// TIA Portal V19 export
// export: Created 2024-12-12T07:14:05.7970126Z, ExportSetting WithDefaults, DisplayName Totally Integrated Automation Portal, DisplayVersion V19 Update 1, DisplayName TIA Portal Openness, DisplayVersion V19 Update 1, DisplayName TIA Portal Version Control Interface, DisplayVersion V19, DisplayName SINAMICS Startdrive Advanced, DisplayVersion V19, DisplayName SINAMICS DCC, DisplayVersion V19, DisplayName SINAMICS Startdrive G130, G150, S120, S150, SINAMICS MV, G220, S200, S210, DisplayVersion V19, DisplayName SINAMICS Startdrive G110M, G120, G120C, G120D, G120P, G115D, DisplayVersion V19, DisplayName STEP 7 Professional, DisplayVersion V19 Update 1, DisplayName STEP 7 Safety, DisplayVersion V19 Update 1, DisplayName WinCC Advanced, DisplayVersion V19 Update 1, DisplayName WinCC Advanced / Unified PC, DisplayVersion V19 Update 1
DATA_BLOCK "AC1"   // DB1013
{ S7_Optimized_Access := 'TRUE' }
VERSION : 0.1
// stored: AutoNumber true, DBAccessibleFromOPCUA true, DBAccessibleFromWebserver true, InstanceOfName EM_AC120_1_2CG, InstanceOfType UDT, IsOnlyStoredInLoadMemory false, IsWriteProtectedInAS false
"EM_AC120_1_2CG"
   // VAR RETAIN
   //    Std : "EM_Std";
   //    Gen : "EM_AC120_1_2CG_Gen";
   //    Param : "EM_AC120_1_2CG_Param";
   //    LastHmiDataParam : "EM_AC120_1_2CG_Param";
   //    Alm : "EM_AC120_1_2CG_Alm";
   //    Sign : "EM_AC120_1_2CG_Sign";
   //    Input : "AC_Input";
   //    Output : "AC_Output";
   //    Ons : "AC_Ons";
   //    "Step" : "AC_Step";
   //    CamCalc : "EM_AC120_1_2CG_CamCalc";
   //    ExchangeFromChain : "EM_AC120_1_2CG_Exchange_FromChain";
   //    ExchangeToChain : "EM_AC120_1_2CG_Exchange_ToChain";
   //    Asc : "EM_AC120_1_2CG_Asc";
   //    Desc : "AC_AscDesc";
   //    Transfer : "EM_AC120_1_2CG_Transfer";
   //    VMaster : "EM_AC120_1_2CG_Virtual";
   //    ThermalReg1 : "AC_ThermalReg";
   //    ShiftUp : Array[0..127] of "TypeMouldData";
   //    ShiftTransfer : Array[0..127] of "TypeMouldData";
   //    ShiftDwn : Array[0..127] of "TypeMouldData";
   // END_VAR
BEGIN
   Std.Cfg_ModuleSync := TRUE;
   Std.Cfg_0_BelongShort_1_BelongLong := TRUE;
   Std.Cfg_ExternalCPU := FALSE;
   Std.Cfg_0_JogWord_1_JogBit := TRUE;
   Std._0_PriorityAlm_1_FirstAlm := FALSE;
   Std.AbortAlmOk := TRUE;
   Std.ServicesAbortAlmOk := TRUE;
   Std.SignOK := TRUE;
   Std.AlmReset := FALSE;
   Std.SignReset := FALSE;
   Std.NewAlm := FALSE;
   Std.NewSign := FALSE;
   Std.RstNewAlm := FALSE;
   Std.RstNewSign := FALSE;
   Std.AllowCopyByCategory := TRUE;
   Std.ForceCopyAll := FALSE;
   Std.InitCategories := FALSE;
   Std.InitCauses := FALSE;
   Std.Diag_AlmFound := FALSE;
   Std.Diag_SignFound := FALSE;
   Std.ScOk := FALSE;
   Std.OkToStop := TRUE;
   Std.PwrDrv := TRUE;
   Std.DriveRunCmd := FALSE;
   Std.ManAct := FALSE;
   Std.MachineSelected := TRUE;
   Std.MachineExtracted := FALSE;
   Std.LocalAbortReq := FALSE;
   Std.CondOkToEnaStaReq := FALSE;
   Std.EnaReq := FALSE;
   Std.EnaStaReq := FALSE;
   Std.StaReq := FALSE;
   Std.ReqStart := FALSE;
   Std.ReqStop := FALSE;
   Std.ReqAbort := TRUE;
   Std.ReqExecute := FALSE;
   Std.ReqReset := FALSE;
   Std.ReqSuspend := FALSE;
   Std.ReqUnSuspend := FALSE;
   Std.StrobeDeviceDiag := FALSE;
   Std.StrobeInverterDiag := FALSE;
   Std.DeviceDiagnosticDone := FALSE;
   Std.InverterDiagnosticDone := FALSE;
   Std.RecipeOnlineLoadDone := FALSE;
   Std.RecipeOnlineSaveDone := FALSE;
   Std.RecipeOfflineLoadDone := FALSE;
   Std.RecipeOfflineSaveDone := FALSE;
   Std.LastHmiDataLoadDone := FALSE;
   Std.LastHmiDataSaveDone := FALSE;
   Std.SummAlmTimeoutStart := FALSE;
   Std.SirenEna := FALSE;
   Std.VisEnButtons := TRUE;
   Std.VisManButtons := FALSE;
   Std.VisHomeButtons := FALSE;
   Std.VisEnButtonsRunning := TRUE;
   Std.Ena_Suspended := TRUE;
   Std.BluStkLgh_Steady_Cond := FALSE;
   Std.BluStkLgh_Frequency1_Cond := FALSE;
   Std.Siren_Frequency4_Cond := FALSE;
   Std.Cfg_ModuleNumber := 4;
   Std.Cfg_DeviceDiagCounter_Preset := 1;
   Std.Cfg_InverterDiagCounter_Preset := 1;
   Std.Cfg_Num_AlmDint := 11;
   Std.Cfg_Num_SignDint := 4;
   Std.Cfg_StaPbt := 65535;
   Std.Cfg_StoPbt := 65535;
   Std.Cfg_RstPbt := -1;
   Std.Cfg_EnaPbt := 65535;
   Std.Cfg_Siren := 1;
   Std.Cfg_Stack := 1;
   Std.Cfg_DisableStates[0..31] := 0;
   Std.Cfg_ModeTransitions[0..31] := 0;
   Std.Cfg_ModeNames[0..31] := '';
   Std.ModeCurrentName := 'Production';
   Std.StateCurrentName := 'Aborted';
   Std.DeviceDiagCounter := 0;
   Std.InverterDiagCounter := 0;
   Std.MaintenanceActivated."0" := FALSE;
   Std.MaintenanceActivated."1" := FALSE;
   Std.MaintenanceActivated."2" := FALSE;
   Std.MaintenanceActivated."3" := FALSE;
   Std.MaintenanceActivated."4" := FALSE;
   Std.MaintenanceActivated."5" := FALSE;
   Std.MaintenanceActivated."6" := FALSE;
   Std.MaintenanceActivated."7" := FALSE;
   Std.MaintenanceActivated."8" := FALSE;
   Std.MaintenanceActivated."9" := FALSE;
   Std.MaintenanceActivated."10" := FALSE;
   Std.MaintenanceActivated."11" := FALSE;
   Std.MaintenanceActivated."12" := FALSE;
   Std.MaintenanceActivated."13" := FALSE;
   Std.MaintenanceActivated."14" := FALSE;
   Std.MaintenanceActivated."15" := FALSE;
   Std.MaintenanceActivated."16" := FALSE;
   Std.MaintenanceActivated."17" := FALSE;
   Std.MaintenanceActivated."18" := FALSE;
   Std.MaintenanceActivated."19" := FALSE;
   Std.MaintenanceActivated."20" := FALSE;
   Std.MaintenanceActivated."21" := FALSE;
   Std.MaintenanceActivated."22" := FALSE;
   Std.MaintenanceActivated."23" := FALSE;
   Std.MaintenanceActivated."24" := FALSE;
   Std.MaintenanceActivated."25" := FALSE;
   Std.MaintenanceActivated."26" := FALSE;
   Std.MaintenanceActivated."27" := FALSE;
   Std.MaintenanceActivated."28" := FALSE;
   Std.MaintenanceActivated."29" := FALSE;
   Std.MaintenanceActivated."30" := FALSE;
   Std.MaintenanceActivated."31" := FALSE;
   Std.MaintenanceReq."0" := FALSE;
   Std.MaintenanceReq."1" := FALSE;
   Std.MaintenanceReq."2" := FALSE;
   Std.MaintenanceReq."3" := FALSE;
   Std.MaintenanceReq."4" := FALSE;
   Std.MaintenanceReq."5" := FALSE;
   Std.MaintenanceReq."6" := FALSE;
   Std.MaintenanceReq."7" := FALSE;
   Std.MaintenanceReq."8" := FALSE;
   Std.MaintenanceReq."9" := FALSE;
   Std.MaintenanceReq."10" := FALSE;
   Std.MaintenanceReq."11" := FALSE;
   Std.MaintenanceReq."12" := FALSE;
   Std.MaintenanceReq."13" := FALSE;
   Std.MaintenanceReq."14" := FALSE;
   Std.MaintenanceReq."15" := FALSE;
   Std.MaintenanceReq."16" := FALSE;
   Std.MaintenanceReq."17" := FALSE;
   Std.MaintenanceReq."18" := FALSE;
   Std.MaintenanceReq."19" := FALSE;
   Std.MaintenanceReq."20" := FALSE;
   Std.MaintenanceReq."21" := FALSE;
   Std.MaintenanceReq."22" := FALSE;
   Std.MaintenanceReq."23" := FALSE;
   Std.MaintenanceReq."24" := FALSE;
   Std.MaintenanceReq."25" := FALSE;
   Std.MaintenanceReq."26" := FALSE;
   Std.MaintenanceReq."27" := FALSE;
   Std.MaintenanceReq."28" := FALSE;
   Std.MaintenanceReq."29" := FALSE;
   Std.MaintenanceReq."30" := FALSE;
   Std.MaintenanceReq."31" := FALSE;
   Std.WithinScreenRange := 0;
   Std.ExchangeToGlobal.Communication.RunMode := FALSE;
   Std.ExchangeToGlobal.Communication.ConnectionFaulted := FALSE;
   Std.ExchangeToGlobal.Gen.Communication := FALSE;
   Std.ExchangeToGlobal.Gen.Selected := TRUE;
   Std.ExchangeToGlobal.Gen.Extracted := FALSE;
   Std.ExchangeToGlobal.Gen.EnaReq := FALSE;
   Std.ExchangeToGlobal.Gen.StaReq := FALSE;
   Std.ExchangeToGlobal.Gen.Started := FALSE;
   Std.ExchangeToGlobal.Gen.Unsuspended := FALSE;
   Std.ExchangeToGlobal.Gen.Ena_Suspended := TRUE;
   Std.ExchangeToGlobal.Gen.sts_Starting := FALSE;
   Std.ExchangeToGlobal.Gen.sts_Stopping := FALSE;
   Std.ExchangeToGlobal.Gen.sts_Aborting := FALSE;
   Std.ExchangeToGlobal.Gen.sts_Suspending := FALSE;
   Std.ExchangeToGlobal.Gen.sts_Unsuspending := FALSE;
   Std.ExchangeToGlobal.Gen.sts_Execute := FALSE;
   Std.ExchangeToGlobal.Gen.sts_Idle := FALSE;
   Std.ExchangeToGlobal.Gen.sts_Stopped := FALSE;
   Std.ExchangeToGlobal.Gen.sts_Aborted := TRUE;
   Std.ExchangeToGlobal.Gen.sts_Suspended := FALSE;
   Std.ExchangeToGlobal.Gen.sts_ModeManual := FALSE;
   Std.ExchangeToGlobal.Gen.sts_ModeAutomatic := TRUE;
   Std.ExchangeToGlobal.Gen.NewAlm := FALSE;
   Std.ExchangeToGlobal.Gen.NewSign := FALSE;
   Std.ExchangeToGlobal.Gen.RecipeOnlineLoadDone := FALSE;
   Std.ExchangeToGlobal.Gen.RecipeOnlineSaveDone := FALSE;
   Std.ExchangeToGlobal.Gen.RecipeOfflineLoadDone := FALSE;
   Std.ExchangeToGlobal.Gen.RecipeOfflineSaveDone := FALSE;
   Std.ExchangeToGlobal.Gen.LastHmiDataLoadDone := FALSE;
   Std.ExchangeToGlobal.Gen.LastHmiDataSaveDone := FALSE;
   Std.ExchangeToGlobal.Gen.InverterDiagnosticDone := FALSE;
   Std.ExchangeToGlobal.Gen.AxisGroupSync := TRUE;
   Std.ExchangeToGlobal.Gen.CmdMode := 1;
   Std.ExchangeToGlobal.Gen.Mode := 1;
   Std.ExchangeToGlobal.Gen.DisableEnaPbt := 0;
   Std.ExchangeToGlobal.Input.StaPbt := FALSE;
   Std.ExchangeToGlobal.Input.StoPbt := FALSE;
   Std.ExchangeToGlobal.Input.RstPbt := FALSE;
   Std.ExchangeToGlobal.Input.EnaPbt := FALSE;
   Std.ExchangeToGlobal.Input._4 := FALSE;
   Std.ExchangeToGlobal.Input._5 := FALSE;
   Std.ExchangeToGlobal.Input._6 := FALSE;
   Std.ExchangeToGlobal.Input._7 := FALSE;
   Std.ExchangeToGlobal.Input._8 := FALSE;
   Std.ExchangeToGlobal.Input._9 := FALSE;
   Std.ExchangeToGlobal.Input._10 := FALSE;
   Std.ExchangeToGlobal.Input._11 := FALSE;
   Std.ExchangeToGlobal.Input._12 := FALSE;
   Std.ExchangeToGlobal.Input._13 := FALSE;
   Std.ExchangeToGlobal.Input._14 := FALSE;
   Std.ExchangeToGlobal.Input._15 := FALSE;
   Std.ExchangeToGlobal.AlmOk.ThSwitch := TRUE;
   Std.ExchangeToGlobal.AlmOk.SafeComm := TRUE;
   Std.ExchangeToGlobal.AlmOk.SafeEmg := TRUE;
   Std.ExchangeToGlobal.AlmOk.SafeGuards := TRUE;
   Std.ExchangeToGlobal.AlmOk.GtaAirGroup := TRUE;
   Std.ExchangeToGlobal.AlmOk.Major := TRUE;
   Std.ExchangeToGlobal.AlmOk.Minor := TRUE;
   Std.ExchangeToGlobal.AlmOk.Spare07 := TRUE;
   Std.ExchangeToGlobal.AlmOk.Spare08 := TRUE;
   Std.ExchangeToGlobal.AlmOk.Spare09 := TRUE;
   Std.ExchangeToGlobal.AlmOk.Spare10 := TRUE;
   Std.ExchangeToGlobal.AlmOk.Spare11 := TRUE;
   Std.ExchangeToGlobal.AlmOk.Spare12 := TRUE;
   Std.ExchangeToGlobal.AlmOk.Spare13 := TRUE;
   Std.ExchangeToGlobal.AlmOk.Spare14 := TRUE;
   Std.ExchangeToGlobal.AlmOk.Spare15 := TRUE;
   Std.ExchangeToGlobal.AlmOk.Spare16 := TRUE;
   Std.ExchangeToGlobal.AlmOk.Spare17 := TRUE;
   Std.ExchangeToGlobal.AlmOk.Spare18 := TRUE;
   Std.ExchangeToGlobal.AlmOk.Spare19 := TRUE;
   Std.ExchangeToGlobal.AlmOk.Spare20 := TRUE;
   Std.ExchangeToGlobal.AlmOk.Spare21 := TRUE;
   Std.ExchangeToGlobal.AlmOk.Spare22 := TRUE;
   Std.ExchangeToGlobal.AlmOk.Spare23 := TRUE;
   Std.ExchangeToGlobal.AlmOk.Spare24 := TRUE;
   Std.ExchangeToGlobal.AlmOk.Spare25 := TRUE;
   Std.ExchangeToGlobal.AlmOk.Spare26 := TRUE;
   Std.ExchangeToGlobal.AlmOk.Spare27 := TRUE;
   Std.ExchangeToGlobal.AlmOk.Spare28 := TRUE;
   Std.ExchangeToGlobal.AlmOk.Spare29 := TRUE;
   Std.ExchangeToGlobal.AlmOk.Spare30 := TRUE;
   Std.ExchangeToGlobal.AlmOk.Spare31 := TRUE;
   Std.ExchangeToGlobal.AlmCauseOk.Ope := TRUE;
   Std.ExchangeToGlobal.AlmCauseOk.Ust := TRUE;
   Std.ExchangeToGlobal.AlmCauseOk.Dst := TRUE;
   Std.ExchangeToGlobal.AlmCauseOk.Ext := TRUE;
   Std.ExchangeToGlobal.AlmCauseOk.Mac := TRUE;
   Std.ExchangeToGlobal.AlmCauseOk.Spare05 := TRUE;
   Std.ExchangeToGlobal.AlmCauseOk.Spare06 := TRUE;
   Std.ExchangeToGlobal.AlmCauseOk.Spare07 := TRUE;
   Std.ExchangeToGlobal.AlmCauseOk.Spare08 := TRUE;
   Std.ExchangeToGlobal.AlmCauseOk.Spare09 := TRUE;
   Std.ExchangeToGlobal.AlmCauseOk.Spare10 := TRUE;
   Std.ExchangeToGlobal.AlmCauseOk.Spare11 := TRUE;
   Std.ExchangeToGlobal.AlmCauseOk.Spare12 := TRUE;
   Std.ExchangeToGlobal.AlmCauseOk.Spare13 := TRUE;
   Std.ExchangeToGlobal.AlmCauseOk.Spare14 := TRUE;
   Std.ExchangeToGlobal.AlmCauseOk.Spare15 := TRUE;
   Std.ExchangeToGlobal.AlmCauseOk.Spare16 := TRUE;
   Std.ExchangeToGlobal.AlmCauseOk.Spare17 := TRUE;
   Std.ExchangeToGlobal.AlmCauseOk.Spare18 := TRUE;
   Std.ExchangeToGlobal.AlmCauseOk.Spare19 := TRUE;
   Std.ExchangeToGlobal.AlmCauseOk.Spare20 := TRUE;
   Std.ExchangeToGlobal.AlmCauseOk.Spare21 := TRUE;
   Std.ExchangeToGlobal.AlmCauseOk.Spare22 := TRUE;
   Std.ExchangeToGlobal.AlmCauseOk.Spare23 := TRUE;
   Std.ExchangeToGlobal.AlmCauseOk.Spare24 := TRUE;
   Std.ExchangeToGlobal.AlmCauseOk.Spare25 := TRUE;
   Std.ExchangeToGlobal.AlmCauseOk.Spare26 := TRUE;
   Std.ExchangeToGlobal.AlmCauseOk.Spare27 := TRUE;
   Std.ExchangeToGlobal.AlmCauseOk.Spare28 := TRUE;
   Std.ExchangeToGlobal.AlmCauseOk.Spare29 := TRUE;
   Std.ExchangeToGlobal.AlmCauseOk.Spare30 := TRUE;
   Std.ExchangeToGlobal.AlmCauseOk.Spare31 := TRUE;
   Std.ExchangeToGlobal.AlmBannerFbk.FirstAlmDetection := FALSE;
   Std.ExchangeToGlobal.AlmBannerFbk.AlmPriority := 100;
   Std.ExchangeToGlobal.AlmBannerFbk.AlmCategory := -1;
   Std.ExchangeToGlobal.AlmBannerFbk.AlmCause := -1;
   Std.ExchangeToGlobal.AlmBannerFbk.AlmID := -1;
   Std.ExchangeToGlobal.AlmBannerFbk.GlobalAbsTime := 0;
   Std.ExchangeToGlobal.SignBannerFbk.SignPriority := 100;
   Std.ExchangeToGlobal.SignBannerFbk.SignCategory := -1;
   Std.ExchangeToGlobal.SignBannerFbk.SignID := -1;
   Std.ExchangeToGlobal.ExtCPU.PushButton.StaPbt := FALSE;
   Std.ExchangeToGlobal.ExtCPU.PushButton.StoPbt := FALSE;
   Std.ExchangeToGlobal.ExtCPU.PushButton.RstPbt := FALSE;
   Std.ExchangeToGlobal.ExtCPU.PushButton.EnaPbt := FALSE;
   Std.ExchangeToGlobal.ExtCPU.PushButton.EnaReq := FALSE;
   Std.ExchangeToGlobal.ExtCPU.PushButton.EnaStaReq := FALSE;
   Std.ExchangeToGlobal.ExtCPU.DeviceDiagDone := FALSE;
   Std.ExchangeToGlobal.ExtCPU.InverterDiagDone := FALSE;
   Std.ExchangeToGlobal.LightSiren.Cfg_StaPbt := 65535;
   Std.ExchangeToGlobal.LightSiren.Cfg_RstPbt := -1;
   Std.ExchangeToGlobal.LightSiren.Cfg_EnaPbt := 65535;
   Std.ExchangeToGlobal.LightSiren.Cfg_Siren := 1;
   Std.ExchangeToGlobal.LightSiren.Cfg_Stack := 1;
   Std.ExchangeToGlobal.LightSiren.Steady.StaPbtLgh := FALSE;
   Std.ExchangeToGlobal.LightSiren.Steady.RstPbtLgh := FALSE;
   Std.ExchangeToGlobal.LightSiren.Steady.EnaPbtLgh := FALSE;
   Std.ExchangeToGlobal.LightSiren.Steady.Siren := FALSE;
   Std.ExchangeToGlobal.LightSiren.Steady.YelStkLgh := FALSE;
   Std.ExchangeToGlobal.LightSiren.Steady.BluStkLgh := FALSE;
   Std.ExchangeToGlobal.LightSiren.Steady.GrnStkLgh := FALSE;
   Std.ExchangeToGlobal.LightSiren.Steady.WhtStkLgh := FALSE;
   Std.ExchangeToGlobal.LightSiren.Steady.Cust1_StaPbtLgh := FALSE;
   Std.ExchangeToGlobal.LightSiren.Steady.Cust1_RstPbtLgh := FALSE;
   Std.ExchangeToGlobal.LightSiren.Steady.Cust1_Siren := FALSE;
   Std.ExchangeToGlobal.LightSiren.Steady.Cust1_RedStkLgh := FALSE;
   Std.ExchangeToGlobal.LightSiren.Steady.Cust1_OngStkLgh := FALSE;
   Std.ExchangeToGlobal.LightSiren.Steady.Cust1_GrnStkLgh := FALSE;
   Std.ExchangeToGlobal.LightSiren.Steady.Cust1_BluStkLgh := FALSE;
   Std.ExchangeToGlobal.LightSiren.Steady.Cust1_WhtStkLgh := FALSE;
   Std.ExchangeToGlobal.LightSiren.Frequency1.StaPbtLgh := FALSE;
   Std.ExchangeToGlobal.LightSiren.Frequency1.RstPbtLgh := FALSE;
   Std.ExchangeToGlobal.LightSiren.Frequency1.EnaPbtLgh := FALSE;
   Std.ExchangeToGlobal.LightSiren.Frequency1.Siren := FALSE;
   Std.ExchangeToGlobal.LightSiren.Frequency1.YelStkLgh := FALSE;
   Std.ExchangeToGlobal.LightSiren.Frequency1.BluStkLgh := FALSE;
   Std.ExchangeToGlobal.LightSiren.Frequency1.GrnStkLgh := FALSE;
   Std.ExchangeToGlobal.LightSiren.Frequency1.WhtStkLgh := FALSE;
   Std.ExchangeToGlobal.LightSiren.Frequency1.Cust1_StaPbtLgh := FALSE;
   Std.ExchangeToGlobal.LightSiren.Frequency1.Cust1_RstPbtLgh := FALSE;
   Std.ExchangeToGlobal.LightSiren.Frequency1.Cust1_Siren := FALSE;
   Std.ExchangeToGlobal.LightSiren.Frequency1.Cust1_RedStkLgh := FALSE;
   Std.ExchangeToGlobal.LightSiren.Frequency1.Cust1_OngStkLgh := FALSE;
   Std.ExchangeToGlobal.LightSiren.Frequency1.Cust1_GrnStkLgh := FALSE;
   Std.ExchangeToGlobal.LightSiren.Frequency1.Cust1_BluStkLgh := FALSE;
   Std.ExchangeToGlobal.LightSiren.Frequency1.Cust1_WhtStkLgh := FALSE;
   Std.ExchangeToGlobal.LightSiren.Frequency2.StaPbtLgh := FALSE;
   Std.ExchangeToGlobal.LightSiren.Frequency2.RstPbtLgh := FALSE;
   Std.ExchangeToGlobal.LightSiren.Frequency2.EnaPbtLgh := FALSE;
   Std.ExchangeToGlobal.LightSiren.Frequency2.Siren := FALSE;
   Std.ExchangeToGlobal.LightSiren.Frequency2.YelStkLgh := FALSE;
   Std.ExchangeToGlobal.LightSiren.Frequency2.BluStkLgh := FALSE;
   Std.ExchangeToGlobal.LightSiren.Frequency2.GrnStkLgh := FALSE;
   Std.ExchangeToGlobal.LightSiren.Frequency2.WhtStkLgh := FALSE;
   Std.ExchangeToGlobal.LightSiren.Frequency2.Cust1_StaPbtLgh := FALSE;
   Std.ExchangeToGlobal.LightSiren.Frequency2.Cust1_RstPbtLgh := FALSE;
   Std.ExchangeToGlobal.LightSiren.Frequency2.Cust1_Siren := FALSE;
   Std.ExchangeToGlobal.LightSiren.Frequency2.Cust1_RedStkLgh := FALSE;
   Std.ExchangeToGlobal.LightSiren.Frequency2.Cust1_OngStkLgh := FALSE;
   Std.ExchangeToGlobal.LightSiren.Frequency2.Cust1_GrnStkLgh := FALSE;
   Std.ExchangeToGlobal.LightSiren.Frequency2.Cust1_BluStkLgh := FALSE;
   Std.ExchangeToGlobal.LightSiren.Frequency2.Cust1_WhtStkLgh := FALSE;
   Std.ExchangeToGlobal.LightSiren.Frequency3.StaPbtLgh := FALSE;
   Std.ExchangeToGlobal.LightSiren.Frequency3.RstPbtLgh := FALSE;
   Std.ExchangeToGlobal.LightSiren.Frequency3.EnaPbtLgh := FALSE;
   Std.ExchangeToGlobal.LightSiren.Frequency3.Siren := FALSE;
   Std.ExchangeToGlobal.LightSiren.Frequency3.YelStkLgh := FALSE;
   Std.ExchangeToGlobal.LightSiren.Frequency3.BluStkLgh := FALSE;
   Std.ExchangeToGlobal.LightSiren.Frequency3.GrnStkLgh := FALSE;
   Std.ExchangeToGlobal.LightSiren.Frequency3.WhtStkLgh := FALSE;
   Std.ExchangeToGlobal.LightSiren.Frequency3.Cust1_StaPbtLgh := FALSE;
   Std.ExchangeToGlobal.LightSiren.Frequency3.Cust1_RstPbtLgh := FALSE;
   Std.ExchangeToGlobal.LightSiren.Frequency3.Cust1_Siren := FALSE;
   Std.ExchangeToGlobal.LightSiren.Frequency3.Cust1_RedStkLgh := FALSE;
   Std.ExchangeToGlobal.LightSiren.Frequency3.Cust1_OngStkLgh := FALSE;
   Std.ExchangeToGlobal.LightSiren.Frequency3.Cust1_GrnStkLgh := FALSE;
   Std.ExchangeToGlobal.LightSiren.Frequency3.Cust1_BluStkLgh := FALSE;
   Std.ExchangeToGlobal.LightSiren.Frequency3.Cust1_WhtStkLgh := FALSE;
   Std.ExchangeToGlobal.LightSiren.Frequency4.StaPbtLgh := FALSE;
   Std.ExchangeToGlobal.LightSiren.Frequency4.RstPbtLgh := FALSE;
   Std.ExchangeToGlobal.LightSiren.Frequency4.EnaPbtLgh := FALSE;
   Std.ExchangeToGlobal.LightSiren.Frequency4.Siren := FALSE;
   Std.ExchangeToGlobal.LightSiren.Frequency4.YelStkLgh := FALSE;
   Std.ExchangeToGlobal.LightSiren.Frequency4.BluStkLgh := FALSE;
   Std.ExchangeToGlobal.LightSiren.Frequency4.GrnStkLgh := FALSE;
   Std.ExchangeToGlobal.LightSiren.Frequency4.WhtStkLgh := FALSE;
   Std.ExchangeToGlobal.LightSiren.Frequency4.Cust1_StaPbtLgh := FALSE;
   Std.ExchangeToGlobal.LightSiren.Frequency4.Cust1_RstPbtLgh := FALSE;
   Std.ExchangeToGlobal.LightSiren.Frequency4.Cust1_Siren := FALSE;
   Std.ExchangeToGlobal.LightSiren.Frequency4.Cust1_RedStkLgh := FALSE;
   Std.ExchangeToGlobal.LightSiren.Frequency4.Cust1_OngStkLgh := FALSE;
   Std.ExchangeToGlobal.LightSiren.Frequency4.Cust1_GrnStkLgh := FALSE;
   Std.ExchangeToGlobal.LightSiren.Frequency4.Cust1_BluStkLgh := FALSE;
   Std.ExchangeToGlobal.LightSiren.Frequency4.Cust1_WhtStkLgh := FALSE;
   Std.ExchangeToGlobal.PackML.Sts_Aborted := TRUE;
   Std.ExchangeToGlobal.PackML.Sts_Aborting := FALSE;
   Std.ExchangeToGlobal.PackML.Sts_Clearing := FALSE;
   Std.ExchangeToGlobal.PackML.Sts_Complete := FALSE;
   Std.ExchangeToGlobal.PackML.Sts_Completing := FALSE;
   Std.ExchangeToGlobal.PackML.Sts_Execute := FALSE;
   Std.ExchangeToGlobal.PackML.Sts_Held := FALSE;
   Std.ExchangeToGlobal.PackML.Sts_Holding := FALSE;
   Std.ExchangeToGlobal.PackML.Sts_Idle := FALSE;
   Std.ExchangeToGlobal.PackML.Sts_Resetting := FALSE;
   Std.ExchangeToGlobal.PackML.Sts_Starting := FALSE;
   Std.ExchangeToGlobal.PackML.Sts_Stopped := FALSE;
   Std.ExchangeToGlobal.PackML.Sts_Stopping := FALSE;
   Std.ExchangeToGlobal.PackML.Sts_Suspended := FALSE;
   Std.ExchangeToGlobal.PackML.Sts_Suspending := FALSE;
   Std.ExchangeToGlobal.PackML.Sts_UnHolding := FALSE;
   Std.ExchangeToGlobal.PackML.Sts_UnSuspending := FALSE;
   Std.ExchangeToGlobal.PackML.Sts_AbortedEnabled := TRUE;
   Std.ExchangeToGlobal.PackML.Sts_AbortingEnabled := TRUE;
   Std.ExchangeToGlobal.PackML.Sts_ClearingEnabled := TRUE;
   Std.ExchangeToGlobal.PackML.Sts_CompleteEnabled := FALSE;
   Std.ExchangeToGlobal.PackML.Sts_CompletingEnabled := FALSE;
   Std.ExchangeToGlobal.PackML.Sts_ExecuteEnabled := TRUE;
   Std.ExchangeToGlobal.PackML.Sts_HeldEnabled := FALSE;
   Std.ExchangeToGlobal.PackML.Sts_HoldingEnabled := FALSE;
   Std.ExchangeToGlobal.PackML.Sts_IdleEnabled := TRUE;
   Std.ExchangeToGlobal.PackML.Sts_ResettingEnabled := TRUE;
   Std.ExchangeToGlobal.PackML.Sts_StartingEnabled := TRUE;
   Std.ExchangeToGlobal.PackML.Sts_StoppedEnabled := TRUE;
   Std.ExchangeToGlobal.PackML.Sts_StoppingEnabled := TRUE;
   Std.ExchangeToGlobal.PackML.Sts_SuspendedEnabled := TRUE;
   Std.ExchangeToGlobal.PackML.Sts_SuspendingEnabled := TRUE;
   Std.ExchangeToGlobal.PackML.Sts_UnHoldingEnabled := FALSE;
   Std.ExchangeToGlobal.PackML.Sts_UnSuspendingEnabled := TRUE;
   Std.ExchangeToGlobal.SignOk := TRUE;
   Std.ExchangeToGlobal."Dint"[0..4] := 0;
   Std.VisAlmTypeBool.ThSwitch := FALSE;
   Std.VisAlmTypeBool.SafeComm := FALSE;
   Std.VisAlmTypeBool.SafeEmg := FALSE;
   Std.VisAlmTypeBool.SafeGuards := TRUE;
   Std.VisAlmTypeBool.GtaAirGroup := FALSE;
   Std.VisAlmTypeBool.Major := FALSE;
   Std.VisAlmTypeBool.Minor := FALSE;
   Std.VisAlmTypeBool.Spare07 := FALSE;
   Std.VisAlmTypeBool.Spare08 := FALSE;
   Std.VisAlmTypeBool.Spare09 := FALSE;
   Std.VisAlmTypeBool.Spare10 := FALSE;
   Std.VisAlmTypeBool.Spare11 := FALSE;
   Std.VisAlmTypeBool.Spare12 := FALSE;
   Std.VisAlmTypeBool.Spare13 := FALSE;
   Std.VisAlmTypeBool.Spare14 := FALSE;
   Std.VisAlmTypeBool.Spare15 := FALSE;
   Std.VisAlmTypeBool.Spare16 := FALSE;
   Std.VisAlmTypeBool.Spare17 := FALSE;
   Std.VisAlmTypeBool.Spare18 := FALSE;
   Std.VisAlmTypeBool.Spare19 := FALSE;
   Std.VisAlmTypeBool.Spare20 := FALSE;
   Std.VisAlmTypeBool.Spare21 := FALSE;
   Std.VisAlmTypeBool.Spare22 := FALSE;
   Std.VisAlmTypeBool.Spare23 := FALSE;
   Std.VisAlmTypeBool.Spare24 := FALSE;
   Std.VisAlmTypeBool.Spare25 := FALSE;
   Std.VisAlmTypeBool.Spare26 := FALSE;
   Std.VisAlmTypeBool.Spare27 := FALSE;
   Std.VisAlmTypeBool.Spare28 := FALSE;
   Std.VisAlmTypeBool.Spare29 := FALSE;
   Std.VisAlmTypeBool.Spare30 := FALSE;
   Std.VisAlmTypeBool.Spare31 := FALSE;
   Std.AlmTypeFbk.ThSwitch := FALSE;
   Std.AlmTypeFbk.SafeComm := FALSE;
   Std.AlmTypeFbk.SafeEmg := FALSE;
   Std.AlmTypeFbk.SafeGuards := FALSE;
   Std.AlmTypeFbk.GtaAirGroup := FALSE;
   Std.AlmTypeFbk.Major := FALSE;
   Std.AlmTypeFbk.Minor := FALSE;
   Std.AlmTypeFbk.Spare07 := FALSE;
   Std.AlmTypeFbk.Spare08 := FALSE;
   Std.AlmTypeFbk.Spare09 := FALSE;
   Std.AlmTypeFbk.Spare10 := FALSE;
   Std.AlmTypeFbk.Spare11 := FALSE;
   Std.AlmTypeFbk.Spare12 := FALSE;
   Std.AlmTypeFbk.Spare13 := FALSE;
   Std.AlmTypeFbk.Spare14 := FALSE;
   Std.AlmTypeFbk.Spare15 := FALSE;
   Std.AlmTypeFbk.Spare16 := FALSE;
   Std.AlmTypeFbk.Spare17 := FALSE;
   Std.AlmTypeFbk.Spare18 := FALSE;
   Std.AlmTypeFbk.Spare19 := FALSE;
   Std.AlmTypeFbk.Spare20 := FALSE;
   Std.AlmTypeFbk.Spare21 := FALSE;
   Std.AlmTypeFbk.Spare22 := FALSE;
   Std.AlmTypeFbk.Spare23 := FALSE;
   Std.AlmTypeFbk.Spare24 := FALSE;
   Std.AlmTypeFbk.Spare25 := FALSE;
   Std.AlmTypeFbk.Spare26 := FALSE;
   Std.AlmTypeFbk.Spare27 := FALSE;
   Std.AlmTypeFbk.Spare28 := FALSE;
   Std.AlmTypeFbk.Spare29 := FALSE;
   Std.AlmTypeFbk.Spare30 := FALSE;
   Std.AlmTypeFbk.Spare31 := FALSE;
   Std.AlmTypeOk.ThSwitch := TRUE;
   Std.AlmTypeOk.SafeComm := TRUE;
   Std.AlmTypeOk.SafeEmg := TRUE;
   Std.AlmTypeOk.SafeGuards := TRUE;
   Std.AlmTypeOk.GtaAirGroup := TRUE;
   Std.AlmTypeOk.Major := TRUE;
   Std.AlmTypeOk.Minor := TRUE;
   Std.AlmTypeOk.Spare07 := TRUE;
   Std.AlmTypeOk.Spare08 := TRUE;
   Std.AlmTypeOk.Spare09 := TRUE;
   Std.AlmTypeOk.Spare10 := TRUE;
   Std.AlmTypeOk.Spare11 := TRUE;
   Std.AlmTypeOk.Spare12 := TRUE;
   Std.AlmTypeOk.Spare13 := TRUE;
   Std.AlmTypeOk.Spare14 := TRUE;
   Std.AlmTypeOk.Spare15 := TRUE;
   Std.AlmTypeOk.Spare16 := TRUE;
   Std.AlmTypeOk.Spare17 := TRUE;
   Std.AlmTypeOk.Spare18 := TRUE;
   Std.AlmTypeOk.Spare19 := TRUE;
   Std.AlmTypeOk.Spare20 := TRUE;
   Std.AlmTypeOk.Spare21 := TRUE;
   Std.AlmTypeOk.Spare22 := TRUE;
   Std.AlmTypeOk.Spare23 := TRUE;
   Std.AlmTypeOk.Spare24 := TRUE;
   Std.AlmTypeOk.Spare25 := TRUE;
   Std.AlmTypeOk.Spare26 := TRUE;
   Std.AlmTypeOk.Spare27 := TRUE;
   Std.AlmTypeOk.Spare28 := TRUE;
   Std.AlmTypeOk.Spare29 := TRUE;
   Std.AlmTypeOk.Spare30 := TRUE;
   Std.AlmTypeOk.Spare31 := TRUE;
   Std.AlmCauseFbk.Ope := FALSE;
   Std.AlmCauseFbk.Ust := FALSE;
   Std.AlmCauseFbk.Dst := FALSE;
   Std.AlmCauseFbk.Ext := FALSE;
   Std.AlmCauseFbk.Mac := FALSE;
   Std.AlmCauseFbk.Spare05 := FALSE;
   Std.AlmCauseFbk.Spare06 := FALSE;
   Std.AlmCauseFbk.Spare07 := FALSE;
   Std.AlmCauseFbk.Spare08 := FALSE;
   Std.AlmCauseFbk.Spare09 := FALSE;
   Std.AlmCauseFbk.Spare10 := FALSE;
   Std.AlmCauseFbk.Spare11 := FALSE;
   Std.AlmCauseFbk.Spare12 := FALSE;
   Std.AlmCauseFbk.Spare13 := FALSE;
   Std.AlmCauseFbk.Spare14 := FALSE;
   Std.AlmCauseFbk.Spare15 := FALSE;
   Std.AlmCauseFbk.Spare16 := FALSE;
   Std.AlmCauseFbk.Spare17 := FALSE;
   Std.AlmCauseFbk.Spare18 := FALSE;
   Std.AlmCauseFbk.Spare19 := FALSE;
   Std.AlmCauseFbk.Spare20 := FALSE;
   Std.AlmCauseFbk.Spare21 := FALSE;
   Std.AlmCauseFbk.Spare22 := FALSE;
   Std.AlmCauseFbk.Spare23 := FALSE;
   Std.AlmCauseFbk.Spare24 := FALSE;
   Std.AlmCauseFbk.Spare25 := FALSE;
   Std.AlmCauseFbk.Spare26 := FALSE;
   Std.AlmCauseFbk.Spare27 := FALSE;
   Std.AlmCauseFbk.Spare28 := FALSE;
   Std.AlmCauseFbk.Spare29 := FALSE;
   Std.AlmCauseFbk.Spare30 := FALSE;
   Std.AlmCauseFbk.Spare31 := FALSE;
   Std.AlmCauseOk.Ope := TRUE;
   Std.AlmCauseOk.Ust := TRUE;
   Std.AlmCauseOk.Dst := TRUE;
   Std.AlmCauseOk.Ext := TRUE;
   Std.AlmCauseOk.Mac := TRUE;
   Std.AlmCauseOk.Spare05 := TRUE;
   Std.AlmCauseOk.Spare06 := TRUE;
   Std.AlmCauseOk.Spare07 := TRUE;
   Std.AlmCauseOk.Spare08 := TRUE;
   Std.AlmCauseOk.Spare09 := TRUE;
   Std.AlmCauseOk.Spare10 := TRUE;
   Std.AlmCauseOk.Spare11 := TRUE;
   Std.AlmCauseOk.Spare12 := TRUE;
   Std.AlmCauseOk.Spare13 := TRUE;
   Std.AlmCauseOk.Spare14 := TRUE;
   Std.AlmCauseOk.Spare15 := TRUE;
   Std.AlmCauseOk.Spare16 := TRUE;
   Std.AlmCauseOk.Spare17 := TRUE;
   Std.AlmCauseOk.Spare18 := TRUE;
   Std.AlmCauseOk.Spare19 := TRUE;
   Std.AlmCauseOk.Spare20 := TRUE;
   Std.AlmCauseOk.Spare21 := TRUE;
   Std.AlmCauseOk.Spare22 := TRUE;
   Std.AlmCauseOk.Spare23 := TRUE;
   Std.AlmCauseOk.Spare24 := TRUE;
   Std.AlmCauseOk.Spare25 := TRUE;
   Std.AlmCauseOk.Spare26 := TRUE;
   Std.AlmCauseOk.Spare27 := TRUE;
   Std.AlmCauseOk.Spare28 := TRUE;
   Std.AlmCauseOk.Spare29 := TRUE;
   Std.AlmCauseOk.Spare30 := TRUE;
   Std.AlmCauseOk.Spare31 := TRUE;
   Std.ForceCategory.ThSwitch := FALSE;
   Std.ForceCategory.SafeComm := TRUE;
   Std.ForceCategory.SafeEmg := TRUE;
   Std.ForceCategory.SafeGuards := FALSE;
   Std.ForceCategory.GtaAirGroup := FALSE;
   Std.ForceCategory.Major := FALSE;
   Std.ForceCategory.Minor := FALSE;
   Std.ForceCategory.Spare07 := FALSE;
   Std.ForceCategory.Spare08 := FALSE;
   Std.ForceCategory.Spare09 := FALSE;
   Std.ForceCategory.Spare10 := FALSE;
   Std.ForceCategory.Spare11 := FALSE;
   Std.ForceCategory.Spare12 := FALSE;
   Std.ForceCategory.Spare13 := FALSE;
   Std.ForceCategory.Spare14 := FALSE;
   Std.ForceCategory.Spare15 := FALSE;
   Std.ForceCategory.Spare16 := FALSE;
   Std.ForceCategory.Spare17 := FALSE;
   Std.ForceCategory.Spare18 := FALSE;
   Std.ForceCategory.Spare19 := FALSE;
   Std.ForceCategory.Spare20 := FALSE;
   Std.ForceCategory.Spare21 := FALSE;
   Std.ForceCategory.Spare22 := FALSE;
   Std.ForceCategory.Spare23 := FALSE;
   Std.ForceCategory.Spare24 := FALSE;
   Std.ForceCategory.Spare25 := FALSE;
   Std.ForceCategory.Spare26 := FALSE;
   Std.ForceCategory.Spare27 := FALSE;
   Std.ForceCategory.Spare28 := FALSE;
   Std.ForceCategory.Spare29 := FALSE;
   Std.ForceCategory.Spare30 := FALSE;
   Std.ForceCategory.Spare31 := FALSE;
   Std.AlmStruct.Alm[0..31] := 0;
   Std.AlmStruct.Category[0..31] := 0;
   Std.AlmStruct.Category[32..63] := 1;
   Std.AlmStruct.Category[64..95] := 2;
   Std.AlmStruct.Category[96..127] := 3;
   Std.AlmStruct.Category[128..159] := 4;
   Std.AlmStruct.Category[160..191] := 5;
   Std.AlmStruct.Category[192..1023] := 6;
   Std.AlmStruct.BannerPriority[0..31] := 0;
   Std.AlmStruct.BannerPriority[32..63] := 1;
   Std.AlmStruct.BannerPriority[64..95] := 2;
   Std.AlmStruct.BannerPriority[96..127] := 3;
   Std.AlmStruct.BannerPriority[128..159] := 4;
   Std.AlmStruct.BannerPriority[160..191] := 5;
   Std.AlmStruct.BannerPriority[192..1023] := 6;
   Std.AlmStruct.Cause[0..63] := 4;
   Std.AlmStruct.Cause[64..127] := 0;
   Std.AlmStruct.Cause[128..159] := 3;
   Std.AlmStruct.Cause[160..206] := 4;
   Std.AlmStruct.Cause[207] := 0;
   Std.AlmStruct.Cause[208..209] := 4;
   Std.AlmStruct.Cause[210] := 0;
   Std.AlmStruct.Cause[211..221] := 4;
   Std.AlmStruct.Cause[222] := 0;
   Std.AlmStruct.Cause[223..324] := 4;
   Std.AlmStruct.Cause[325] := 0;
   Std.AlmStruct.Cause[326..327] := 4;
   Std.AlmStruct.Cause[328] := 0;
   Std.AlmStruct.Cause[329..330] := 4;
   Std.AlmStruct.Cause[331] := 0;
   Std.AlmStruct.Cause[332..333] := 4;
   Std.AlmStruct.Cause[334] := 0;
   Std.AlmStruct.Cause[335..1023] := 4;
   Std.AlmBannerFbk.FirstAlmDetection := FALSE;
   Std.AlmBannerFbk.AlmPriority := 100;
   Std.AlmBannerFbk.AlmCategory := -1;
   Std.AlmBannerFbk.AlmCause := -1;
   Std.AlmBannerFbk.AlmID := -1;
   Std.AlmBannerFbk.GlobalAbsTime := 0;
   Std.SignStruct.Sign[0..31] := 0;
   Std.SignStruct.Category[0..1023] := 0;
   Std.SignStruct.BannerPriority[0..63] := 3;
   Std.SignStruct.BannerPriority[64..95] := 1;
   Std.SignStruct.BannerPriority[96..127] := 2;
   Std.SignStruct.BannerPriority[128..1023] := 0;
   Std.SignBannerFbk.SignPriority := 100;
   Std.SignBannerFbk.SignCategory := -1;
   Std.SignBannerFbk.SignID := -1;
   Std.MaintenanceInput.Clock_1Hz := FALSE;
   Std.MaintenanceInput.CountEnable := FALSE;
   Std.MaintenanceInput.CondToBeActivated := TRUE;
   Std.MaintenanceInput.EventsStrobe := 0;
   Std.LightSiren.Cfg_StaPbt := 65535;
   Std.LightSiren.Cfg_RstPbt := -1;
   Std.LightSiren.Cfg_EnaPbt := 65535;
   Std.LightSiren.Cfg_Siren := 1;
   Std.LightSiren.Cfg_Stack := 1;
   Std.LightSiren.Steady.StaPbtLgh := FALSE;
   Std.LightSiren.Steady.RstPbtLgh := FALSE;
   Std.LightSiren.Steady.EnaPbtLgh := FALSE;
   Std.LightSiren.Steady.Siren := FALSE;
   Std.LightSiren.Steady.YelStkLgh := FALSE;
   Std.LightSiren.Steady.BluStkLgh := FALSE;
   Std.LightSiren.Steady.GrnStkLgh := FALSE;
   Std.LightSiren.Steady.WhtStkLgh := FALSE;
   Std.LightSiren.Steady.Cust1_StaPbtLgh := FALSE;
   Std.LightSiren.Steady.Cust1_RstPbtLgh := FALSE;
   Std.LightSiren.Steady.Cust1_Siren := FALSE;
   Std.LightSiren.Steady.Cust1_RedStkLgh := FALSE;
   Std.LightSiren.Steady.Cust1_OngStkLgh := FALSE;
   Std.LightSiren.Steady.Cust1_GrnStkLgh := FALSE;
   Std.LightSiren.Steady.Cust1_BluStkLgh := FALSE;
   Std.LightSiren.Steady.Cust1_WhtStkLgh := FALSE;
   Std.LightSiren.Frequency1.StaPbtLgh := FALSE;
   Std.LightSiren.Frequency1.RstPbtLgh := FALSE;
   Std.LightSiren.Frequency1.EnaPbtLgh := FALSE;
   Std.LightSiren.Frequency1.Siren := FALSE;
   Std.LightSiren.Frequency1.YelStkLgh := FALSE;
   Std.LightSiren.Frequency1.BluStkLgh := FALSE;
   Std.LightSiren.Frequency1.GrnStkLgh := FALSE;
   Std.LightSiren.Frequency1.WhtStkLgh := FALSE;
   Std.LightSiren.Frequency1.Cust1_StaPbtLgh := FALSE;
   Std.LightSiren.Frequency1.Cust1_RstPbtLgh := FALSE;
   Std.LightSiren.Frequency1.Cust1_Siren := FALSE;
   Std.LightSiren.Frequency1.Cust1_RedStkLgh := FALSE;
   Std.LightSiren.Frequency1.Cust1_OngStkLgh := FALSE;
   Std.LightSiren.Frequency1.Cust1_GrnStkLgh := FALSE;
   Std.LightSiren.Frequency1.Cust1_BluStkLgh := FALSE;
   Std.LightSiren.Frequency1.Cust1_WhtStkLgh := FALSE;
   Std.LightSiren.Frequency2.StaPbtLgh := FALSE;
   Std.LightSiren.Frequency2.RstPbtLgh := FALSE;
   Std.LightSiren.Frequency2.EnaPbtLgh := FALSE;
   Std.LightSiren.Frequency2.Siren := FALSE;
   Std.LightSiren.Frequency2.YelStkLgh := FALSE;
   Std.LightSiren.Frequency2.BluStkLgh := FALSE;
   Std.LightSiren.Frequency2.GrnStkLgh := FALSE;
   Std.LightSiren.Frequency2.WhtStkLgh := FALSE;
   Std.LightSiren.Frequency2.Cust1_StaPbtLgh := FALSE;
   Std.LightSiren.Frequency2.Cust1_RstPbtLgh := FALSE;
   Std.LightSiren.Frequency2.Cust1_Siren := FALSE;
   Std.LightSiren.Frequency2.Cust1_RedStkLgh := FALSE;
   Std.LightSiren.Frequency2.Cust1_OngStkLgh := FALSE;
   Std.LightSiren.Frequency2.Cust1_GrnStkLgh := FALSE;
   Std.LightSiren.Frequency2.Cust1_BluStkLgh := FALSE;
   Std.LightSiren.Frequency2.Cust1_WhtStkLgh := FALSE;
   Std.LightSiren.Frequency3.StaPbtLgh := FALSE;
   Std.LightSiren.Frequency3.RstPbtLgh := FALSE;
   Std.LightSiren.Frequency3.EnaPbtLgh := FALSE;
   Std.LightSiren.Frequency3.Siren := FALSE;
   Std.LightSiren.Frequency3.YelStkLgh := FALSE;
   Std.LightSiren.Frequency3.BluStkLgh := FALSE;
   Std.LightSiren.Frequency3.GrnStkLgh := FALSE;
   Std.LightSiren.Frequency3.WhtStkLgh := FALSE;
   Std.LightSiren.Frequency3.Cust1_StaPbtLgh := FALSE;
   Std.LightSiren.Frequency3.Cust1_RstPbtLgh := FALSE;
   Std.LightSiren.Frequency3.Cust1_Siren := FALSE;
   Std.LightSiren.Frequency3.Cust1_RedStkLgh := FALSE;
   Std.LightSiren.Frequency3.Cust1_OngStkLgh := FALSE;
   Std.LightSiren.Frequency3.Cust1_GrnStkLgh := FALSE;
   Std.LightSiren.Frequency3.Cust1_BluStkLgh := FALSE;
   Std.LightSiren.Frequency3.Cust1_WhtStkLgh := FALSE;
   Std.LightSiren.Frequency4.StaPbtLgh := FALSE;
   Std.LightSiren.Frequency4.RstPbtLgh := FALSE;
   Std.LightSiren.Frequency4.EnaPbtLgh := FALSE;
   Std.LightSiren.Frequency4.Siren := FALSE;
   Std.LightSiren.Frequency4.YelStkLgh := FALSE;
   Std.LightSiren.Frequency4.BluStkLgh := FALSE;
   Std.LightSiren.Frequency4.GrnStkLgh := FALSE;
   Std.LightSiren.Frequency4.WhtStkLgh := FALSE;
   Std.LightSiren.Frequency4.Cust1_StaPbtLgh := FALSE;
   Std.LightSiren.Frequency4.Cust1_RstPbtLgh := FALSE;
   Std.LightSiren.Frequency4.Cust1_Siren := FALSE;
   Std.LightSiren.Frequency4.Cust1_RedStkLgh := FALSE;
   Std.LightSiren.Frequency4.Cust1_OngStkLgh := FALSE;
   Std.LightSiren.Frequency4.Cust1_GrnStkLgh := FALSE;
   Std.LightSiren.Frequency4.Cust1_BluStkLgh := FALSE;
   Std.LightSiren.Frequency4.Cust1_WhtStkLgh := FALSE;
   Std.MachineStateModel.EnableIn := FALSE;
   Std.MachineStateModel.EnableOut := FALSE;
   Std.MachineStateModel.Cmd_Mode := 1;
   Std.MachineStateModel.Cmd_Reset := FALSE;
   Std.MachineStateModel.Cmd_Start := FALSE;
   Std.MachineStateModel.Cmd_Stop := FALSE;
   Std.MachineStateModel.Cmd_Hold := FALSE;
   Std.MachineStateModel.Cmd_UnHold := FALSE;
   Std.MachineStateModel.Cmd_Suspend := FALSE;
   Std.MachineStateModel.Cmd_UnSuspend := FALSE;
   Std.MachineStateModel.Cmd_Abort := FALSE;
   Std.MachineStateModel.Cmd_Clear := FALSE;
   Std.MachineStateModel.Cmd_StateComplete := FALSE;
   Std.MachineStateModel.Cmd_ModeManual := FALSE;
   Std.MachineStateModel.Cmd_ModeProduce := TRUE;
   Std.MachineStateModel.Cfg_RemoteCmdEnable := FALSE;
   Std.MachineStateModel.Inp_RemoteModeCmd := 0;
   Std.MachineStateModel.Inp_RemoteModeCmdChangeRequest := FALSE;
   Std.MachineStateModel.Inp_RemoteStateCmd := 0;
   Std.MachineStateModel.Inp_RemoteStateCmdChangeRequest := FALSE;
   Std.MachineStateModel.StartRequest := FALSE;
   Std.MachineStateModel.ResetRequest := FALSE;
   Std.MachineStateModel.Sts_StateCurrent := 9;
   Std.MachineStateModel.Sts_ModeCurrent := 1;
   Std.MachineStateModel.Sts_DisabledStates := 203776;
   Std.MachineStateModel.Sts_ProductionModeCurrent := TRUE;
   Std.MachineStateModel.Sts_ManualModeCurrent := FALSE;
   Std.MachineStateModel.Sts_ClearingEnabled := TRUE;
   Std.MachineStateModel.Sts_StoppedEnabled := TRUE;
   Std.MachineStateModel.Sts_StartingEnabled := TRUE;
   Std.MachineStateModel.Sts_IdleEnabled := TRUE;
   Std.MachineStateModel.Sts_SuspendedEnabled := TRUE;
   Std.MachineStateModel.Sts_ExecuteEnabled := TRUE;
   Std.MachineStateModel.Sts_StoppingEnabled := TRUE;
   Std.MachineStateModel.Sts_AbortingEnabled := TRUE;
   Std.MachineStateModel.Sts_AbortedEnabled := TRUE;
   Std.MachineStateModel.Sts_HoldingEnabled := FALSE;
   Std.MachineStateModel.Sts_HeldEnabled := FALSE;
   Std.MachineStateModel.Sts_UnHoldingEnabled := FALSE;
   Std.MachineStateModel.Sts_SuspendingEnabled := TRUE;
   Std.MachineStateModel.Sts_UnSuspendingEnabled := TRUE;
   Std.MachineStateModel.Sts_ResettingEnabled := TRUE;
   Std.MachineStateModel.Sts_CompletingEnabled := FALSE;
   Std.MachineStateModel.Sts_CompleteEnabled := FALSE;
   Std.MachineStateModel.Sts_ModeChangeNotAllowed := FALSE;
   Std.MachineStateModel.Sts_Clearing := FALSE;
   Std.MachineStateModel.Sts_Stopped := FALSE;
   Std.MachineStateModel.Sts_Starting := FALSE;
   Std.MachineStateModel.Sts_Idle := FALSE;
   Std.MachineStateModel.Sts_Suspended := FALSE;
   Std.MachineStateModel.Sts_Execute := FALSE;
   Std.MachineStateModel.Sts_Stopping := FALSE;
   Std.MachineStateModel.Sts_Aborting := FALSE;
   Std.MachineStateModel.Sts_Aborted := TRUE;
   Std.MachineStateModel.Sts_Holding := FALSE;
   Std.MachineStateModel.Sts_Held := FALSE;
   Std.MachineStateModel.Sts_UnHolding := FALSE;
   Std.MachineStateModel.Sts_Suspending := FALSE;
   Std.MachineStateModel.Sts_UnSuspending := FALSE;
   Std.MachineStateModel.Sts_Resetting := FALSE;
   Std.MachineStateModel.Sts_Complete := FALSE;
   Std.MachineStateModel.Sts_Completing := FALSE;
   Std.MachineStateModel.Sts_AbortingDone := FALSE;
   Std.MachineStateModel.Sts_ClearingDone := FALSE;
   Std.MachineStateModel.Sts_ResettingDone := FALSE;
   Std.MachineStateModel.Sts_StartingDone := FALSE;
   Std.MachineStateModel.Sts_UnSuspendingDone := FALSE;
   Std.MachineStateModel.Sts_StoppingDone := FALSE;
   Std.MachineStateModel.Sts_SuspendingDone := FALSE;
   Std.MachineStateModel.TON_TimeoutStop.PT := T#0MS;
   Std.MachineStateModel.TON_TimeoutStop.IN := FALSE;
   Std.MachineStateModel.TON_TimeoutAbort.PT := T#0MS;
   Std.MachineStateModel.TON_TimeoutAbort.IN := FALSE;
   Std.MachineStateModel.TON_Start.PT := T#0MS;
   Std.MachineStateModel.TON_Start.IN := FALSE;
   Std.TON_SafetyOn.PT := T#1S;
   Std.TON_SafetyOn.IN := FALSE;
   Std.TOF_SirenEna.PT := T#5S;
   Std.TOF_SirenEna.ET := T#5S;
   Std.TOF_SirenEna.IN := FALSE;
   Gen.Cfg_1Cooler_0Heater := FALSE;
   Gen.AlmOk := TRUE;
   Gen.MotionScOk := FALSE;
   Gen.CycleOn := FALSE;
   Gen.StationEmpty := FALSE;
   Gen.GrtPosReverse := FALSE;
   Gen.RangeLowSpeed := TRUE;
   Gen.Work := FALSE;
   Gen.OutChainObstruction := TRUE;
   Gen.MotionOkToStop := TRUE;
   Gen.ManCmdBefReverseStep := FALSE;
   Gen.ManCmdReverseStep := FALSE;
   Gen.AxisCammingStart := FALSE;
   Gen.AuxAxisCamRequest := FALSE;
   Gen.InitPos := TRUE;
   Gen.InitPosAxis := TRUE;
   Gen.CamHookAxis := FALSE;
   Gen.DrivesEnabled := FALSE;
   Gen.SlowFirstStepAfterEmerg := FALSE;
   Gen.ManMovMemory := FALSE;
   Gen.MemFirstStep_IP := FALSE;
   Gen.ManConsoleSelection := 0;
   Gen.Mould_Counter := 0;
   Gen.Cfg_Mould_ChainSteps_Asc := 1;
   Gen.Cfg_Mould_ChainSteps_Desc := 2;
   Gen.Cfg_Mould_TransferSteps := 1;
   Gen.Cfg_Mould_ColumnCapacity_Asc := 60;
   Gen.Cfg_Mould_ColumnCapacity_Desc := 120;
   Gen.Cfg_Mould_TransferCapacity := 9;
   Gen.Cfg_Mould_EndPos := 0;
   Gen.Shift_ColumnLenght_Asc := 61;
   Gen.Shift_ColumnLenght_Desc := 122;
   Gen.RTO_Work.PT := T#1M;
   Gen.RTO_Work.ET := T#0MS;
   Gen.RTO_Work.IN := FALSE;
   Gen.TON_ScOK.PT := T#20S;
   Gen.TON_ScOK.IN := FALSE;
   Gen.TON_TimeoutWork.PT := T#20S;
   Gen.TON_TimeoutWork.IN := FALSE;
   Gen.TON_DelayVirtualCommandOFF.PT := T#200MS;
   Gen.TON_DelayVirtualCommandOFF.ET := T#200MS;
   Gen.TON_DelayVirtualCommandOFF.IN := FALSE;
   Gen.TON_AlmMouOnLug_InfOpeSid.PT := T#100MS;
   Gen.TON_AlmMouOnLug_InfOpeSid.IN := FALSE;
   Gen.TON_AlmMouOnLug_InfNotOpeSid.PT := T#100MS;
   Gen.TON_AlmMouOnLug_InfNotOpeSid.IN := FALSE;
   Gen.TON_AlmMouOnLug_OufOpeSid.PT := T#100MS;
   Gen.TON_AlmMouOnLug_OufOpeSid.IN := FALSE;
   Gen.TON_AlmMouOnLug_OufNotOpeSid.PT := T#100MS;
   Gen.TON_AlmMouOnLug_OufNotOpeSid.IN := FALSE;
   Param.Gen_Ena := TRUE;
   Param.Asc_Torque_Limit := 20.0;
   Param.Desc_Torque_Limit := 20.0;
   Param.Transfer_Torque_Limit := 35.0;
   Param.ThermalReg1_Ena := FALSE;
   Param.ThermalReg1_Ena_Fan1 := TRUE;
   Param.ThermalReg1_Ena_Fan2 := TRUE;
   Param.ThermalReg1_Ena_Fan3 := TRUE;
   Param.ThermalReg1_Ena_Fan4 := TRUE;
   Param.ThermalReg1_Ena_Fan5 := TRUE;
   Param.ThermalReg1_Ena_Fan6 := TRUE;
   Param.ThermalReg1_WorkingTemperature := 10.0;
   Param.ThermalReg1_StoppingTemperature := 10.0;
   Param.ThermalReg1_LongStopTemperature := 10.0;
   Param.ThermalReg1_WorkingFanSpeed := 30.0;
   Param.ThermalReg1_StoppingFanSpeed := 30.0;
   Param.ThermalReg1_LongStopFanSpeed := 10.0;
   Param.ThermalReg1_LongStopDelay := 20;
   Param.ThermalReg1_RecircValveManSetpoint := 0.0;
   Param.ThermalReg1_HeatExchValveManSetpoint := 0.0;
   Param.ThermalReg1_PumpSpeed := 45.0;
   LastHmiDataParam.Gen_Ena := FALSE;
   LastHmiDataParam.Asc_Torque_Limit := 0.0;
   LastHmiDataParam.Desc_Torque_Limit := 0.0;
   LastHmiDataParam.Transfer_Torque_Limit := 0.0;
   LastHmiDataParam.ThermalReg1_Ena := FALSE;
   LastHmiDataParam.ThermalReg1_Ena_Fan1 := FALSE;
   LastHmiDataParam.ThermalReg1_Ena_Fan2 := FALSE;
   LastHmiDataParam.ThermalReg1_Ena_Fan3 := FALSE;
   LastHmiDataParam.ThermalReg1_Ena_Fan4 := FALSE;
   LastHmiDataParam.ThermalReg1_Ena_Fan5 := FALSE;
   LastHmiDataParam.ThermalReg1_Ena_Fan6 := FALSE;
   LastHmiDataParam.ThermalReg1_WorkingTemperature := 0.0;
   LastHmiDataParam.ThermalReg1_StoppingTemperature := 0.0;
   LastHmiDataParam.ThermalReg1_LongStopTemperature := 0.0;
   LastHmiDataParam.ThermalReg1_WorkingFanSpeed := 0.0;
   LastHmiDataParam.ThermalReg1_StoppingFanSpeed := 0.0;
   LastHmiDataParam.ThermalReg1_LongStopFanSpeed := 0.0;
   LastHmiDataParam.ThermalReg1_LongStopDelay := 0;
   LastHmiDataParam.ThermalReg1_RecircValveManSetpoint := 0.0;
   LastHmiDataParam.ThermalReg1_HeatExchValveManSetpoint := 0.0;
   LastHmiDataParam.ThermalReg1_PumpSpeed := 0.0;
   Alm.ThSwitch."0" := FALSE;   // AC1.Alm.ThSwitch.0
   Alm.ThSwitch."1" := FALSE;   // AC1.Alm.ThSwitch.1
   Alm.ThSwitch."2" := FALSE;   // AC1.Alm.ThSwitch.2
   Alm.ThSwitch."3" := FALSE;   // AC1.Alm.ThSwitch.3
   Alm.ThSwitch."4" := FALSE;   // AC1.Alm.ThSwitch.4
   Alm.ThSwitch."5" := FALSE;   // AC1.Alm.ThSwitch.5
   Alm.ThSwitch."6" := FALSE;   // AC1.Alm.ThSwitch.6
   Alm.ThSwitch."7" := FALSE;   // AC1.Alm.ThSwitch.7
   Alm.ThSwitch."8" := FALSE;   // AC1.Alm.ThSwitch.8
   Alm.ThSwitch."9" := FALSE;   // AC1.Alm.ThSwitch.9
   Alm.ThSwitch."10" := FALSE;   // AC1.Alm.ThSwitch.10
   Alm.ThSwitch."11" := FALSE;   // AC1.Alm.ThSwitch.11
   Alm.ThSwitch."12" := FALSE;   // AC1.Alm.ThSwitch.12
   Alm.ThSwitch."13" := FALSE;   // AC1.Alm.ThSwitch.13
   Alm.ThSwitch."14" := FALSE;   // AC1.Alm.ThSwitch.14
   Alm.ThSwitch."15" := FALSE;   // AC1.Alm.ThSwitch.15
   Alm.ThSwitch."16" := FALSE;   // AC1.Alm.ThSwitch.16
   Alm.ThSwitch."17" := FALSE;   // AC1.Alm.ThSwitch.17
   Alm.ThSwitch."18" := FALSE;   // AC1.Alm.ThSwitch.18
   Alm.ThSwitch."19" := FALSE;   // AC1.Alm.ThSwitch.19
   Alm.ThSwitch."20" := FALSE;   // AC1.Alm.ThSwitch.20
   Alm.ThSwitch."21" := FALSE;   // AC1.Alm.ThSwitch.21
   Alm.ThSwitch."22" := FALSE;   // AC1.Alm.ThSwitch.22
   Alm.ThSwitch."23" := FALSE;   // AC1.Alm.ThSwitch.23
   Alm.ThSwitch."24" := FALSE;   // AC1.Alm.ThSwitch.24
   Alm.ThSwitch."25" := FALSE;   // AC1.Alm.ThSwitch.25
   Alm.ThSwitch."26" := FALSE;   // AC1.Alm.ThSwitch.26
   Alm.ThSwitch."27" := FALSE;   // AC1.Alm.ThSwitch.27
   Alm.ThSwitch."28" := FALSE;   // AC1.Alm.ThSwitch.28
   Alm.ThSwitch."29" := FALSE;   // AC1.Alm.ThSwitch.29
   Alm.ThSwitch."30" := FALSE;   // AC1.Alm.ThSwitch.30
   Alm.ThSwitch."31" := FALSE;   // AC1.Alm.ThSwitch.31
   Alm.SafeComm."0" := FALSE;   // AC1.Alm.SafeComm.0 > Communication fault point_io zone AC1 in (1AC300FK3)
   Alm.SafeComm."1" := FALSE;   // AC1.Alm.SafeComm.1
   Alm.SafeComm."2" := FALSE;   // AC1.Alm.SafeComm.2
   Alm.SafeComm."3" := FALSE;   // AC1.Alm.SafeComm.3
   Alm.SafeComm."4" := FALSE;   // AC1.Alm.SafeComm.4
   Alm.SafeComm."5" := FALSE;   // AC1.Alm.SafeComm.5
   Alm.SafeComm."6" := FALSE;   // AC1.Alm.SafeComm.6
   Alm.SafeComm."7" := FALSE;   // AC1.Alm.SafeComm.7
   Alm.SafeComm."8" := FALSE;   // AC1.Alm.SafeComm.8
   Alm.SafeComm."9" := FALSE;   // AC1.Alm.SafeComm.9
   Alm.SafeComm."10" := FALSE;   // AC1.Alm.SafeComm.10 > Communication fault simotion ascent (1AC40TB5)
   Alm.SafeComm."11" := FALSE;   // AC1.Alm.SafeComm.11 > Communication fault simotion transfer (1AC40TB5)
   Alm.SafeComm."12" := FALSE;   // AC1.Alm.SafeComm.12 > Communication fault simotion descent (1AC42TB5)
   Alm.SafeComm."13" := FALSE;   // AC1.Alm.SafeComm.13
   Alm.SafeComm."14" := FALSE;   // AC1.Alm.SafeComm.14
   Alm.SafeComm."15" := FALSE;   // AC1.Alm.SafeComm.15
   Alm.SafeComm."16" := FALSE;   // AC1.Alm.SafeComm.16
   Alm.SafeComm."17" := FALSE;   // AC1.Alm.SafeComm.17
   Alm.SafeComm."18" := FALSE;   // AC1.Alm.SafeComm.18
   Alm.SafeComm."19" := FALSE;   // AC1.Alm.SafeComm.19
   Alm.SafeComm."20" := FALSE;   // AC1.Alm.SafeComm.20
   Alm.SafeComm."21" := FALSE;   // AC1.Alm.SafeComm.21
   Alm.SafeComm."22" := FALSE;   // AC1.Alm.SafeComm.22
   Alm.SafeComm."23" := FALSE;   // AC1.Alm.SafeComm.23
   Alm.SafeComm."24" := FALSE;   // AC1.Alm.SafeComm.24
   Alm.SafeComm."25" := FALSE;   // AC1.Alm.SafeComm.25
   Alm.SafeComm."26" := FALSE;   // AC1.Alm.SafeComm.26
   Alm.SafeComm."27" := FALSE;   // AC1.Alm.SafeComm.27
   Alm.SafeComm."28" := FALSE;   // AC1.Alm.SafeComm.28
   Alm.SafeComm."29" := FALSE;   // AC1.Alm.SafeComm.29
   Alm.SafeComm."30" := FALSE;   // AC1.Alm.SafeComm.30
   Alm.SafeComm."31" := FALSE;   // AC1.Alm.SafeComm.31
   Alm.SafeEmg."0" := FALSE;   // AC1.Alm.SafeEmg.0 > Emergency pressed jog air conditioning (1AC370SF2)
   Alm.SafeEmg."1" := FALSE;   // AC1.Alm.SafeEmg.1
   Alm.SafeEmg."2" := FALSE;   // AC1.Alm.SafeEmg.2
   Alm.SafeEmg."3" := FALSE;   // AC1.Alm.SafeEmg.3
   Alm.SafeEmg."4" := FALSE;   // AC1.Alm.SafeEmg.4
   Alm.SafeEmg."5" := FALSE;   // AC1.Alm.SafeEmg.5
   Alm.SafeEmg."6" := FALSE;   // AC1.Alm.SafeEmg.6
   Alm.SafeEmg."7" := FALSE;   // AC1.Alm.SafeEmg.7
   Alm.SafeEmg."8" := FALSE;   // AC1.Alm.SafeEmg.8
   Alm.SafeEmg."9" := FALSE;   // AC1.Alm.SafeEmg.9
   Alm.SafeEmg."10" := FALSE;   // AC1.Alm.SafeEmg.10
   Alm.SafeEmg."11" := FALSE;   // AC1.Alm.SafeEmg.11
   Alm.SafeEmg."12" := FALSE;   // AC1.Alm.SafeEmg.12
   Alm.SafeEmg."13" := FALSE;   // AC1.Alm.SafeEmg.13
   Alm.SafeEmg."14" := FALSE;   // AC1.Alm.SafeEmg.14
   Alm.SafeEmg."15" := FALSE;   // AC1.Alm.SafeEmg.15
   Alm.SafeEmg."16" := FALSE;   // AC1.Alm.SafeEmg.16 > Instruction fault emergency stop jog (1AC370SF2)
   Alm.SafeEmg."17" := FALSE;   // AC1.Alm.SafeEmg.17
   Alm.SafeEmg."18" := FALSE;   // AC1.Alm.SafeEmg.18
   Alm.SafeEmg."19" := FALSE;   // AC1.Alm.SafeEmg.19
   Alm.SafeEmg."20" := FALSE;   // AC1.Alm.SafeEmg.20
   Alm.SafeEmg."21" := FALSE;   // AC1.Alm.SafeEmg.21
   Alm.SafeEmg."22" := FALSE;   // AC1.Alm.SafeEmg.22
   Alm.SafeEmg."23" := FALSE;   // AC1.Alm.SafeEmg.23
   Alm.SafeEmg."24" := FALSE;   // AC1.Alm.SafeEmg.24
   Alm.SafeEmg."25" := FALSE;   // AC1.Alm.SafeEmg.25
   Alm.SafeEmg."26" := FALSE;   // AC1.Alm.SafeEmg.26
   Alm.SafeEmg."27" := FALSE;   // AC1.Alm.SafeEmg.27
   Alm.SafeEmg."28" := FALSE;   // AC1.Alm.SafeEmg.28
   Alm.SafeEmg."29" := FALSE;   // AC1.Alm.SafeEmg.29
   Alm.SafeEmg."30" := FALSE;   // AC1.Alm.SafeEmg.30
   Alm.SafeEmg."31" := FALSE;   // AC1.Alm.SafeEmg.31
   Alm.SafeGuards."0" := FALSE;   // AC1.Alm.SafeGuards.0 > Safe guard operator side open (1AC115FQ3A/4A)
   Alm.SafeGuards."1" := FALSE;   // AC1.Alm.SafeGuards.1 > Safe guard not operator side open (1AC115FQ3/4)
   Alm.SafeGuards."2" := FALSE;   // AC1.Alm.SafeGuards.2
   Alm.SafeGuards."3" := FALSE;   // AC1.Alm.SafeGuards.3
   Alm.SafeGuards."4" := FALSE;   // AC1.Alm.SafeGuards.4
   Alm.SafeGuards."5" := FALSE;   // AC1.Alm.SafeGuards.5
   Alm.SafeGuards."6" := FALSE;   // AC1.Alm.SafeGuards.6
   Alm.SafeGuards."7" := FALSE;   // AC1.Alm.SafeGuards.7
   Alm.SafeGuards."8" := FALSE;   // AC1.Alm.SafeGuards.8
   Alm.SafeGuards."9" := FALSE;   // AC1.Alm.SafeGuards.9
   Alm.SafeGuards."10" := FALSE;   // AC1.Alm.SafeGuards.10
   Alm.SafeGuards."11" := FALSE;   // AC1.Alm.SafeGuards.11
   Alm.SafeGuards."12" := FALSE;   // AC1.Alm.SafeGuards.12
   Alm.SafeGuards."13" := FALSE;   // AC1.Alm.SafeGuards.13
   Alm.SafeGuards."14" := FALSE;   // AC1.Alm.SafeGuards.14
   Alm.SafeGuards."15" := FALSE;   // AC1.Alm.SafeGuards.15
   Alm.SafeGuards."16" := FALSE;   // AC1.Alm.SafeGuards.16 > Module fault (1AC370KF1)
   Alm.SafeGuards."17" := FALSE;   // AC1.Alm.SafeGuards.17
   Alm.SafeGuards."18" := FALSE;   // AC1.Alm.SafeGuards.18
   Alm.SafeGuards."19" := FALSE;   // AC1.Alm.SafeGuards.19
   Alm.SafeGuards."20" := FALSE;   // AC1.Alm.SafeGuards.20
   Alm.SafeGuards."21" := FALSE;   // AC1.Alm.SafeGuards.21
   Alm.SafeGuards."22" := FALSE;   // AC1.Alm.SafeGuards.22 > Drive ascent fault (1AC40MA8)
   Alm.SafeGuards."23" := FALSE;   // AC1.Alm.SafeGuards.23 > Drive transfer fault (1AC41MA8)
   Alm.SafeGuards."24" := FALSE;   // AC1.Alm.SafeGuards.24 > Drive descent fault (1AC42MA8)
   Alm.SafeGuards."25" := FALSE;   // AC1.Alm.SafeGuards.25
   Alm.SafeGuards."26" := FALSE;   // AC1.Alm.SafeGuards.26 > Termal regulation inverter recirculation pump fault (1AC60TB6)
   Alm.SafeGuards."27" := FALSE;   // AC1.Alm.SafeGuards.27
   Alm.SafeGuards."28" := FALSE;   // AC1.Alm.SafeGuards.28
   Alm.SafeGuards."29" := FALSE;   // AC1.Alm.SafeGuards.29
   Alm.SafeGuards."30" := FALSE;   // AC1.Alm.SafeGuards.30
   Alm.SafeGuards."31" := FALSE;   // AC1.Alm.SafeGuards.31
   Alm.GtaAirGroup."0" := FALSE;   // AC1.Alm.GtaAirGroup.0
   Alm.GtaAirGroup."1" := FALSE;   // AC1.Alm.GtaAirGroup.1
   Alm.GtaAirGroup."2" := FALSE;   // AC1.Alm.GtaAirGroup.2
   Alm.GtaAirGroup."3" := FALSE;   // AC1.Alm.GtaAirGroup.3
   Alm.GtaAirGroup."4" := FALSE;   // AC1.Alm.GtaAirGroup.4
   Alm.GtaAirGroup."5" := FALSE;   // AC1.Alm.GtaAirGroup.5
   Alm.GtaAirGroup."6" := FALSE;   // AC1.Alm.GtaAirGroup.6
   Alm.GtaAirGroup."7" := FALSE;   // AC1.Alm.GtaAirGroup.7
   Alm.GtaAirGroup."8" := FALSE;   // AC1.Alm.GtaAirGroup.8
   Alm.GtaAirGroup."9" := FALSE;   // AC1.Alm.GtaAirGroup.9
   Alm.GtaAirGroup."10" := FALSE;   // AC1.Alm.GtaAirGroup.10
   Alm.GtaAirGroup."11" := FALSE;   // AC1.Alm.GtaAirGroup.11
   Alm.GtaAirGroup."12" := FALSE;   // AC1.Alm.GtaAirGroup.12
   Alm.GtaAirGroup."13" := FALSE;   // AC1.Alm.GtaAirGroup.13
   Alm.GtaAirGroup."14" := FALSE;   // AC1.Alm.GtaAirGroup.14
   Alm.GtaAirGroup."15" := FALSE;   // AC1.Alm.GtaAirGroup.15
   Alm.GtaAirGroup."16" := FALSE;   // AC1.Alm.GtaAirGroup.16
   Alm.GtaAirGroup."17" := FALSE;   // AC1.Alm.GtaAirGroup.17
   Alm.GtaAirGroup."18" := FALSE;   // AC1.Alm.GtaAirGroup.18
   Alm.GtaAirGroup."19" := FALSE;   // AC1.Alm.GtaAirGroup.19
   Alm.GtaAirGroup."20" := FALSE;   // AC1.Alm.GtaAirGroup.20
   Alm.GtaAirGroup."21" := FALSE;   // AC1.Alm.GtaAirGroup.21
   Alm.GtaAirGroup."22" := FALSE;   // AC1.Alm.GtaAirGroup.22
   Alm.GtaAirGroup."23" := FALSE;   // AC1.Alm.GtaAirGroup.23
   Alm.GtaAirGroup."24" := FALSE;   // AC1.Alm.GtaAirGroup.24
   Alm.GtaAirGroup."25" := FALSE;   // AC1.Alm.GtaAirGroup.25
   Alm.GtaAirGroup."26" := FALSE;   // AC1.Alm.GtaAirGroup.26
   Alm.GtaAirGroup."27" := FALSE;   // AC1.Alm.GtaAirGroup.27
   Alm.GtaAirGroup."28" := FALSE;   // AC1.Alm.GtaAirGroup.28
   Alm.GtaAirGroup."29" := FALSE;   // AC1.Alm.GtaAirGroup.29
   Alm.GtaAirGroup."30" := FALSE;   // AC1.Alm.GtaAirGroup.30
   Alm.GtaAirGroup."31" := FALSE;   // AC1.Alm.GtaAirGroup.31
   Alm.Major."0" := FALSE;   // AC1.Alm.Major.0
   Alm.Major."1" := FALSE;   // AC1.Alm.Major.1 > Instruction fault dead man safety button (1AC370SF2)
   Alm.Major."2" := FALSE;   // AC1.Alm.Major.2 > Instruction fault ascent simotion safe limited speed
   Alm.Major."3" := FALSE;   // AC1.Alm.Major.3 > Instruction fault transfer simotion safe limited speed
   Alm.Major."4" := FALSE;   // AC1.Alm.Major.4 > Instruction fault descent simotion safe limited speed
   Alm.Major."5" := FALSE;   // AC1.Alm.Major.5
   Alm.Major."6" := FALSE;   // AC1.Alm.Major.6
   Alm.Major."7" := FALSE;   // AC1.Alm.Major.7
   Alm.Major."8" := FALSE;   // AC1.Alm.Major.8
   Alm.Major."9" := FALSE;   // AC1.Alm.Major.9
   Alm.Major."10" := FALSE;   // AC1.Alm.Major.10
   Alm.Major."11" := FALSE;   // AC1.Alm.Major.11
   Alm.Major."12" := FALSE;   // AC1.Alm.Major.12
   Alm.Major."13" := FALSE;   // AC1.Alm.Major.13
   Alm.Major."14" := FALSE;   // AC1.Alm.Major.14
   Alm.Major."15" := FALSE;   // AC1.Alm.Major.15
   Alm.Major."16" := FALSE;   // AC1.Alm.Major.16
   Alm.Major."17" := FALSE;   // AC1.Alm.Major.17
   Alm.Major."18" := FALSE;   // AC1.Alm.Major.18
   Alm.Major."19" := FALSE;   // AC1.Alm.Major.19
   Alm.Major."20" := FALSE;   // AC1.Alm.Major.20
   Alm.Major."21" := FALSE;   // AC1.Alm.Major.21
   Alm.Major."22" := FALSE;   // AC1.Alm.Major.22
   Alm.Major."23" := FALSE;   // AC1.Alm.Major.23
   Alm.Major."24" := FALSE;   // AC1.Alm.Major.24
   Alm.Major."25" := FALSE;   // AC1.Alm.Major.25
   Alm.Major."26" := FALSE;   // AC1.Alm.Major.26
   Alm.Major."27" := FALSE;   // AC1.Alm.Major.27
   Alm.Major."28" := FALSE;   // AC1.Alm.Major.28
   Alm.Major."29" := FALSE;   // AC1.Alm.Major.29
   Alm.Major."30" := FALSE;   // AC1.Alm.Major.30
   Alm.Major."31" := FALSE;   // AC1.Alm.Major.31
   Alm.Minor."0" := FALSE;   // AC1.Alm.Minor.0 > Station in manual mode selected
   Alm.Minor."1" := FALSE;   // AC1.Alm.Minor.1 > Timeout movement
   Alm.Minor."2" := FALSE;   // AC1.Alm.Minor.2 > Timeout start condition
   Alm.Minor."3" := FALSE;   // AC1.Alm.Minor.3 > Ascent/descent in chain obstruction
   Alm.Minor."4" := FALSE;   // AC1.Alm.Minor.4
   Alm.Minor."5" := FALSE;   // AC1.Alm.Minor.5 > Jog connector inserted
   Alm.Minor."6" := FALSE;   // AC1.Alm.Minor.6
   Alm.Minor."7" := FALSE;   // AC1.Alm.Minor.7
   Alm.Minor."8" := FALSE;   // AC1.Alm.Minor.8
   Alm.Minor."9" := FALSE;   // AC1.Alm.Minor.9
   Alm.Minor."10" := FALSE;   // AC1.Alm.Minor.10
   Alm.Minor."11" := FALSE;   // AC1.Alm.Minor.11
   Alm.Minor."12" := FALSE;   // AC1.Alm.Minor.12
   Alm.Minor."13" := FALSE;   // AC1.Alm.Minor.13
   Alm.Minor."14" := FALSE;   // AC1.Alm.Minor.14
   Alm.Minor."15" := FALSE;   // AC1.Alm.Minor.15
   Alm.Minor."16" := FALSE;   // AC1.Alm.Minor.16 > Mould between ascent/descent (1AC330BR8)
   Alm.Minor."17" := FALSE;   // AC1.Alm.Minor.17 > Mould on lug infeed cooler not ope side (1AC330BR5)
   Alm.Minor."18" := FALSE;   // AC1.Alm.Minor.18 > Mould on lug infeed cooler ope side (1AC330BR6)
   Alm.Minor."19" := FALSE;   // AC1.Alm.Minor.19 > Mould on lug outfeed cooler not ope side (1AC330BR9)
   Alm.Minor."20" := FALSE;   // AC1.Alm.Minor.20 > Mould on lug outfeed cooler ope side (1AC330BR7)
   Alm.Minor."21" := FALSE;   // AC1.Alm.Minor.21
   Alm.Minor."22" := FALSE;   // AC1.Alm.Minor.22
   Alm.Minor."23" := FALSE;   // AC1.Alm.Minor.23
   Alm.Minor."24" := FALSE;   // AC1.Alm.Minor.24
   Alm.Minor."25" := FALSE;   // AC1.Alm.Minor.25
   Alm.Minor."26" := FALSE;   // AC1.Alm.Minor.26
   Alm.Minor."27" := FALSE;   // AC1.Alm.Minor.27
   Alm.Minor."28" := FALSE;   // AC1.Alm.Minor.28
   Alm.Minor."29" := FALSE;   // AC1.Alm.Minor.29
   Alm.Minor."30" := FALSE;   // AC1.Alm.Minor.30 > Air treatment switched off, please start it from main cabinet
   Alm.Minor."31" := FALSE;   // AC1.Alm.Minor.31
   Alm.MinorAsc."0" := FALSE;   // AC1.Alm.MinorAsc.0 > Ascent not in phase (1AC40MA8)
   Alm.MinorAsc."1" := FALSE;   // AC1.Alm.MinorAsc.1 > Ascent torque limit (1AC40MA8)
   Alm.MinorAsc."2" := FALSE;   // AC1.Alm.MinorAsc.2 > Ascent drive fault (1AC40MA8)
   Alm.MinorAsc."3" := FALSE;   // AC1.Alm.MinorAsc.3 > Ascent loss of zero position (1AC40MA8)
   Alm.MinorAsc."4" := FALSE;   // AC1.Alm.MinorAsc.4
   Alm.MinorAsc."5" := FALSE;   // AC1.Alm.MinorAsc.5 > Ascent safety no ok simotion (1AC40MA8)
   Alm.MinorAsc."6" := FALSE;   // AC1.Alm.MinorAsc.6
   Alm.MinorAsc."7" := FALSE;   // AC1.Alm.MinorAsc.7
   Alm.MinorAsc."8" := FALSE;   // AC1.Alm.MinorAsc.8
   Alm.MinorAsc."9" := FALSE;   // AC1.Alm.MinorAsc.9
   Alm.MinorAsc."10" := FALSE;   // AC1.Alm.MinorAsc.10 > Ascent error cam hooking
   Alm.MinorAsc."11" := FALSE;   // AC1.Alm.MinorAsc.11
   Alm.MinorAsc."12" := FALSE;   // AC1.Alm.MinorAsc.12
   Alm.MinorAsc."13" := FALSE;   // AC1.Alm.MinorAsc.13
   Alm.MinorAsc."14" := FALSE;   // AC1.Alm.MinorAsc.14
   Alm.MinorAsc."15" := FALSE;   // AC1.Alm.MinorAsc.15 > Please phase chain in manual mode
   Alm.MinorAsc."16" := FALSE;   // AC1.Alm.MinorAsc.16
   Alm.MinorAsc."17" := FALSE;   // AC1.Alm.MinorAsc.17
   Alm.MinorAsc."18" := FALSE;   // AC1.Alm.MinorAsc.18
   Alm.MinorAsc."19" := FALSE;   // AC1.Alm.MinorAsc.19
   Alm.MinorAsc."20" := FALSE;   // AC1.Alm.MinorAsc.20 > Safe limit speed exceeded ascent (1AC40TB5)
   Alm.MinorAsc."21" := FALSE;   // AC1.Alm.MinorAsc.21
   Alm.MinorAsc."22" := FALSE;   // AC1.Alm.MinorAsc.22
   Alm.MinorAsc."23" := FALSE;   // AC1.Alm.MinorAsc.23
   Alm.MinorAsc."24" := FALSE;   // AC1.Alm.MinorAsc.24
   Alm.MinorAsc."25" := FALSE;   // AC1.Alm.MinorAsc.25
   Alm.MinorAsc."26" := FALSE;   // AC1.Alm.MinorAsc.26
   Alm.MinorAsc."27" := FALSE;   // AC1.Alm.MinorAsc.27
   Alm.MinorAsc."28" := FALSE;   // AC1.Alm.MinorAsc.28
   Alm.MinorAsc."29" := FALSE;   // AC1.Alm.MinorAsc.29
   Alm.MinorAsc."30" := FALSE;   // AC1.Alm.MinorAsc.30
   Alm.MinorAsc."31" := FALSE;   // AC1.Alm.MinorAsc.31
   Alm.MinorDesc."0" := FALSE;   // AC1.Alm.MinorDesc.0 > Descent not in phase (1AC42MA8)
   Alm.MinorDesc."1" := FALSE;   // AC1.Alm.MinorDesc.1 > Descent torque limit (1AC42MA8)
   Alm.MinorDesc."2" := FALSE;   // AC1.Alm.MinorDesc.2 > Descent drive fault (1AC42MA8)
   Alm.MinorDesc."3" := FALSE;   // AC1.Alm.MinorDesc.3 > Descent loss of zero position (1AC42MA8)
   Alm.MinorDesc."4" := FALSE;   // AC1.Alm.MinorDesc.4
   Alm.MinorDesc."5" := FALSE;   // AC1.Alm.MinorDesc.5 > Descent safety no ok simotion (1AC42MA8)
   Alm.MinorDesc."6" := FALSE;   // AC1.Alm.MinorDesc.6
   Alm.MinorDesc."7" := FALSE;   // AC1.Alm.MinorDesc.7
   Alm.MinorDesc."8" := FALSE;   // AC1.Alm.MinorDesc.8
   Alm.MinorDesc."9" := FALSE;   // AC1.Alm.MinorDesc.9
   Alm.MinorDesc."10" := FALSE;   // AC1.Alm.MinorDesc.10 > Descent error cam hooking
   Alm.MinorDesc."11" := FALSE;   // AC1.Alm.MinorDesc.11
   Alm.MinorDesc."12" := FALSE;   // AC1.Alm.MinorDesc.12
   Alm.MinorDesc."13" := FALSE;   // AC1.Alm.MinorDesc.13
   Alm.MinorDesc."14" := FALSE;   // AC1.Alm.MinorDesc.14
   Alm.MinorDesc."15" := FALSE;   // AC1.Alm.MinorDesc.15 > Please phase chain in manual mode
   Alm.MinorDesc."16" := FALSE;   // AC1.Alm.MinorDesc.16
   Alm.MinorDesc."17" := FALSE;   // AC1.Alm.MinorDesc.17
   Alm.MinorDesc."18" := FALSE;   // AC1.Alm.MinorDesc.18
   Alm.MinorDesc."19" := FALSE;   // AC1.Alm.MinorDesc.19
   Alm.MinorDesc."20" := FALSE;   // AC1.Alm.MinorDesc.20 > Safe limit speed exceeded descent (1AC42TB5)
   Alm.MinorDesc."21" := FALSE;   // AC1.Alm.MinorDesc.21
   Alm.MinorDesc."22" := FALSE;   // AC1.Alm.MinorDesc.22
   Alm.MinorDesc."23" := FALSE;   // AC1.Alm.MinorDesc.23
   Alm.MinorDesc."24" := FALSE;   // AC1.Alm.MinorDesc.24
   Alm.MinorDesc."25" := FALSE;   // AC1.Alm.MinorDesc.25
   Alm.MinorDesc."26" := FALSE;   // AC1.Alm.MinorDesc.26
   Alm.MinorDesc."27" := FALSE;   // AC1.Alm.MinorDesc.27
   Alm.MinorDesc."28" := FALSE;   // AC1.Alm.MinorDesc.28
   Alm.MinorDesc."29" := FALSE;   // AC1.Alm.MinorDesc.29
   Alm.MinorDesc."30" := FALSE;   // AC1.Alm.MinorDesc.30
   Alm.MinorDesc."31" := FALSE;   // AC1.Alm.MinorDesc.31
   Alm.MinorTransfer."0" := FALSE;   // AC1.Alm.MinorTransfer.0 > Transfer not in phase (1AC41MA8)
   Alm.MinorTransfer."1" := FALSE;   // AC1.Alm.MinorTransfer.1 > Transfer torque limit (1AC41MA8)
   Alm.MinorTransfer."2" := FALSE;   // AC1.Alm.MinorTransfer.2 > Transfer drive fault (1AC41MA8)
   Alm.MinorTransfer."3" := FALSE;   // AC1.Alm.MinorTransfer.3 > Transfer loss of zero position (1AC41MA8)
   Alm.MinorTransfer."4" := FALSE;   // AC1.Alm.MinorTransfer.4
   Alm.MinorTransfer."5" := FALSE;   // AC1.Alm.MinorTransfer.5 > Transfer safety no ok simotion (1AC41MA8)
   Alm.MinorTransfer."6" := FALSE;   // AC1.Alm.MinorTransfer.6 > Transfer waiting for operator validation
   Alm.MinorTransfer."7" := FALSE;   // AC1.Alm.MinorTransfer.7 > Transfer slave forward refer to its master
   Alm.MinorTransfer."8" := FALSE;   // AC1.Alm.MinorTransfer.8 > Transfer slave backward refer to its master
   Alm.MinorTransfer."9" := FALSE;   // AC1.Alm.MinorTransfer.9 > Transfer slave unwind refer to its master
   Alm.MinorTransfer."10" := FALSE;   // AC1.Alm.MinorTransfer.10 > Transfer error cam hooking
   Alm.MinorTransfer."11" := FALSE;   // AC1.Alm.MinorTransfer.11 > Execute a single transfer step before restart
   Alm.MinorTransfer."12" := FALSE;   // AC1.Alm.MinorTransfer.12
   Alm.MinorTransfer."13" := FALSE;   // AC1.Alm.MinorTransfer.13
   Alm.MinorTransfer."14" := FALSE;   // AC1.Alm.MinorTransfer.14
   Alm.MinorTransfer."15" := FALSE;   // AC1.Alm.MinorTransfer.15
   Alm.MinorTransfer."16" := FALSE;   // AC1.Alm.MinorTransfer.16
   Alm.MinorTransfer."17" := FALSE;   // AC1.Alm.MinorTransfer.17
   Alm.MinorTransfer."18" := FALSE;   // AC1.Alm.MinorTransfer.18
   Alm.MinorTransfer."19" := FALSE;   // AC1.Alm.MinorTransfer.19
   Alm.MinorTransfer."20" := FALSE;   // AC1.Alm.MinorTransfer.20 > Safe limit speed exceeded transfer (1AC40TB5)
   Alm.MinorTransfer."21" := FALSE;   // AC1.Alm.MinorTransfer.21
   Alm.MinorTransfer."22" := FALSE;   // AC1.Alm.MinorTransfer.22
   Alm.MinorTransfer."23" := FALSE;   // AC1.Alm.MinorTransfer.23
   Alm.MinorTransfer."24" := FALSE;   // AC1.Alm.MinorTransfer.24
   Alm.MinorTransfer."25" := FALSE;   // AC1.Alm.MinorTransfer.25
   Alm.MinorTransfer."26" := FALSE;   // AC1.Alm.MinorTransfer.26
   Alm.MinorTransfer."27" := FALSE;   // AC1.Alm.MinorTransfer.27
   Alm.MinorTransfer."28" := FALSE;   // AC1.Alm.MinorTransfer.28
   Alm.MinorTransfer."29" := FALSE;   // AC1.Alm.MinorTransfer.29
   Alm.MinorTransfer."30" := FALSE;   // AC1.Alm.MinorTransfer.30
   Alm.MinorTransfer."31" := FALSE;   // AC1.Alm.MinorTransfer.31
   Alm.MinorThermalReg1."0" := FALSE;   // AC1.Alm.MinorThermalReg1.0 > Battery 1 - thermal protection recirculation pump (1AC60QA8)
   Alm.MinorThermalReg1."1" := FALSE;   // AC1.Alm.MinorThermalReg1.1 > Battery 1 - not in position
   Alm.MinorThermalReg1."2" := FALSE;   // AC1.Alm.MinorThermalReg1.2 > Battery 1 - cold water ON/OFF valve timeout movement (1AC334BG2/3)
   Alm.MinorThermalReg1."3" := FALSE;   // AC1.Alm.MinorThermalReg1.3 > Battery 1 - thermal protection fan 1 (1AC70QA9)
   Alm.MinorThermalReg1."4" := FALSE;   // AC1.Alm.MinorThermalReg1.4 > Battery 1 - fan 1 not ready (1AC70MA9)
   Alm.MinorThermalReg1."5" := FALSE;   // AC1.Alm.MinorThermalReg1.5 > Battery 1 - fan 1 connector not inserted (1AC332TB2)
   Alm.MinorThermalReg1."6" := FALSE;   // AC1.Alm.MinorThermalReg1.6 > Battery 1 - thermal protection fan 2 (1AC71QA9)
   Alm.MinorThermalReg1."7" := FALSE;   // AC1.Alm.MinorThermalReg1.7 > Battery 1 - fan 2 not ready (1AC71MA9)
   Alm.MinorThermalReg1."8" := FALSE;   // AC1.Alm.MinorThermalReg1.8 > Battery 1 - fan 2 connector not inserted (1AC332TB4)
   Alm.MinorThermalReg1."9" := FALSE;   // AC1.Alm.MinorThermalReg1.9 > Battery 1 - thermal protection fan 3 (1AC72QA9)
   Alm.MinorThermalReg1."10" := FALSE;   // AC1.Alm.MinorThermalReg1.10 > Battery 1 - fan 3 not ready (1AC72MA9)
   Alm.MinorThermalReg1."11" := FALSE;   // AC1.Alm.MinorThermalReg1.11 > Battery 1 - fan 3 connector not inserted (1AC332TB6)
   Alm.MinorThermalReg1."12" := FALSE;   // AC1.Alm.MinorThermalReg1.12 > Battery 1 - thermal protection fan 4 (1AC73QA9)
   Alm.MinorThermalReg1."13" := FALSE;   // AC1.Alm.MinorThermalReg1.13 > Battery 1 - fan 4 not ready (1AC73MA9)
   Alm.MinorThermalReg1."14" := FALSE;   // AC1.Alm.MinorThermalReg1.14 > Battery 1 - fan 4 connector not inserted (1AC332TB8)
   Alm.MinorThermalReg1."15" := FALSE;   // AC1.Alm.MinorThermalReg1.15 > Battery 1 - hot water ON/OFF valve timeout movement (1AC334BG4/5)
   Alm.MinorThermalReg1."16" := FALSE;   // AC1.Alm.MinorThermalReg1.16 > Battery 1 - inverter fault pump (1AC60TB6)
   Alm.MinorThermalReg1."17" := FALSE;   // AC1.Alm.MinorThermalReg1.17 > Battery 1 - communication fault inverter pump (1AC60TB6)
   Alm.MinorThermalReg1."18" := FALSE;   // AC1.Alm.MinorThermalReg1.18 > Battery 1 - air sensor 1 fault (1AC305BT3)
   Alm.MinorThermalReg1."19" := FALSE;   // AC1.Alm.MinorThermalReg1.19 > Battery 1 - air sensor 2 fault (1AC307BT3)
   Alm.MinorThermalReg1."20" := FALSE;   // AC1.Alm.MinorThermalReg1.20 > Battery 1 - water sensor fault (1AC307BT7)
   Alm.MinorThermalReg1."21" := FALSE;   // AC1.Alm.MinorThermalReg1.21 > Battery 1 - infeed water pressure sensor fault (1AC308BP3)
   Alm.MinorThermalReg1."22" := FALSE;   // AC1.Alm.MinorThermalReg1.22 > Battery 1 - outfeed water pressure sensor fault (1AC308BP7)
   Alm.MinorThermalReg1."23" := FALSE;   // AC1.Alm.MinorThermalReg1.23 > Battery 1 - heating liquid temperature too high
   Alm.MinorThermalReg1."24" := FALSE;   // AC1.Alm.MinorThermalReg1.24 > Battery 1 - control valve out of position (1AC320QM3)
   Alm.MinorThermalReg1."25" := FALSE;   // AC1.Alm.MinorThermalReg1.25
   Alm.MinorThermalReg1."26" := FALSE;   // AC1.Alm.MinorThermalReg1.26 > Battery 1 - thermal protection fan 5 (1AC74QA9)
   Alm.MinorThermalReg1."27" := FALSE;   // AC1.Alm.MinorThermalReg1.27 > Battery 1 - fan 5 not ready (1AC74MA9)
   Alm.MinorThermalReg1."28" := FALSE;   // AC1.Alm.MinorThermalReg1.28 > Battery 1 - fan 5 connector not inserted (1AC333TB2)
   Alm.MinorThermalReg1."29" := FALSE;   // AC1.Alm.MinorThermalReg1.29 > Battery 1 - thermal protection fan 6 (1AC75QA9)
   Alm.MinorThermalReg1."30" := FALSE;   // AC1.Alm.MinorThermalReg1.30 > Battery 1 - fan 6 not ready (1AC75MA9)
   Alm.MinorThermalReg1."31" := FALSE;   // AC1.Alm.MinorThermalReg1.31 > Battery 1 - fan 6 connector not inserted (1AC333TB4)
   Sign.General."0" := FALSE;   // AC1.Sign.General.0 > Jog inserted
   Sign.General."1" := FALSE;   // AC1.Sign.General.1
   Sign.General."2" := FALSE;   // AC1.Sign.General.2
   Sign.General."3" := FALSE;   // AC1.Sign.General.3
   Sign.General."4" := FALSE;   // AC1.Sign.General.4
   Sign.General."5" := FALSE;   // AC1.Sign.General.5
   Sign.General."6" := FALSE;   // AC1.Sign.General.6
   Sign.General."7" := FALSE;   // AC1.Sign.General.7
   Sign.General."8" := FALSE;   // AC1.Sign.General.8
   Sign.General."9" := FALSE;   // AC1.Sign.General.9
   Sign.General."10" := FALSE;   // AC1.Sign.General.10
   Sign.General."11" := FALSE;   // AC1.Sign.General.11
   Sign.General."12" := FALSE;   // AC1.Sign.General.12
   Sign.General."13" := FALSE;   // AC1.Sign.General.13
   Sign.General."14" := FALSE;   // AC1.Sign.General.14
   Sign.General."15" := FALSE;   // AC1.Sign.General.15
   Sign.General."16" := FALSE;   // AC1.Sign.General.16
   Sign.General."17" := FALSE;   // AC1.Sign.General.17
   Sign.General."18" := FALSE;   // AC1.Sign.General.18
   Sign.General."19" := FALSE;   // AC1.Sign.General.19
   Sign.General."20" := FALSE;   // AC1.Sign.General.20
   Sign.General."21" := FALSE;   // AC1.Sign.General.21
   Sign.General."22" := FALSE;   // AC1.Sign.General.22
   Sign.General."23" := FALSE;   // AC1.Sign.General.23
   Sign.General."24" := FALSE;   // AC1.Sign.General.24
   Sign.General."25" := FALSE;   // AC1.Sign.General.25
   Sign.General."26" := FALSE;   // AC1.Sign.General.26
   Sign.General."27" := FALSE;   // AC1.Sign.General.27
   Sign.General."28" := FALSE;   // AC1.Sign.General.28
   Sign.General."29" := FALSE;   // AC1.Sign.General.29
   Sign.General."30" := FALSE;   // AC1.Sign.General.30
   Sign.General."31" := FALSE;   // AC1.Sign.General.31
   Sign.ThermalReg1."0" := FALSE;   // AC1.Sign.ThermalReg1.0
   Sign.ThermalReg1."1" := FALSE;   // AC1.Sign.ThermalReg1.1
   Sign.ThermalReg1."2" := FALSE;   // AC1.Sign.ThermalReg1.2
   Sign.ThermalReg1."3" := FALSE;   // AC1.Sign.ThermalReg1.3
   Sign.ThermalReg1."4" := FALSE;   // AC1.Sign.ThermalReg1.4
   Sign.ThermalReg1."5" := FALSE;   // AC1.Sign.ThermalReg1.5
   Sign.ThermalReg1."6" := FALSE;   // AC1.Sign.ThermalReg1.6
   Sign.ThermalReg1."7" := FALSE;   // AC1.Sign.ThermalReg1.7
   Sign.ThermalReg1."8" := FALSE;   // AC1.Sign.ThermalReg1.8
   Sign.ThermalReg1."9" := FALSE;   // AC1.Sign.ThermalReg1.9
   Sign.ThermalReg1."10" := FALSE;   // AC1.Sign.ThermalReg1.10
   Sign.ThermalReg1."11" := FALSE;   // AC1.Sign.ThermalReg1.11
   Sign.ThermalReg1."12" := FALSE;   // AC1.Sign.ThermalReg1.12
   Sign.ThermalReg1."13" := FALSE;   // AC1.Sign.ThermalReg1.13
   Sign.ThermalReg1."14" := FALSE;   // AC1.Sign.ThermalReg1.14
   Sign.ThermalReg1."15" := FALSE;   // AC1.Sign.ThermalReg1.15 > High temperature battery
   Sign.ThermalReg1."16" := FALSE;   // AC1.Sign.ThermalReg1.16 > Low temperature battery
   Sign.ThermalReg1."17" := FALSE;   // AC1.Sign.ThermalReg1.17
   Sign.ThermalReg1."18" := FALSE;   // AC1.Sign.ThermalReg1.18
   Sign.ThermalReg1."19" := FALSE;   // AC1.Sign.ThermalReg1.19
   Sign.ThermalReg1."20" := FALSE;   // AC1.Sign.ThermalReg1.20
   Sign.ThermalReg1."21" := FALSE;   // AC1.Sign.ThermalReg1.21
   Sign.ThermalReg1."22" := FALSE;   // AC1.Sign.ThermalReg1.22
   Sign.ThermalReg1."23" := FALSE;   // AC1.Sign.ThermalReg1.23
   Sign.ThermalReg1."24" := FALSE;   // AC1.Sign.ThermalReg1.24
   Sign.ThermalReg1."25" := FALSE;   // AC1.Sign.ThermalReg1.25
   Sign.ThermalReg1."26" := FALSE;   // AC1.Sign.ThermalReg1.26
   Sign.ThermalReg1."27" := FALSE;   // AC1.Sign.ThermalReg1.27
   Sign.ThermalReg1."28" := FALSE;   // AC1.Sign.ThermalReg1.28
   Sign.ThermalReg1."29" := FALSE;   // AC1.Sign.ThermalReg1.29
   Sign.ThermalReg1."30" := FALSE;   // AC1.Sign.ThermalReg1.30
   Sign.ThermalReg1."31" := FALSE;   // AC1.Sign.ThermalReg1.31
   Sign.Maintenance_Req."0" := FALSE;   // AC1.Sign.Maintenance_Req.0 > Maintenance 0 request
   Sign.Maintenance_Req."1" := FALSE;   // AC1.Sign.Maintenance_Req.1 > Maintenance 1 request
   Sign.Maintenance_Req."2" := FALSE;   // AC1.Sign.Maintenance_Req.2 > Maintenance 2 request
   Sign.Maintenance_Req."3" := FALSE;   // AC1.Sign.Maintenance_Req.3 > Maintenance 3 request
   Sign.Maintenance_Req."4" := FALSE;   // AC1.Sign.Maintenance_Req.4 > Maintenance 4 request
   Sign.Maintenance_Req."5" := FALSE;   // AC1.Sign.Maintenance_Req.5 > Maintenance 5 request
   Sign.Maintenance_Req."6" := FALSE;   // AC1.Sign.Maintenance_Req.6 > Maintenance 6 request
   Sign.Maintenance_Req."7" := FALSE;   // AC1.Sign.Maintenance_Req.7 > Maintenance 7 request
   Sign.Maintenance_Req."8" := FALSE;   // AC1.Sign.Maintenance_Req.8 > Maintenance 8 request
   Sign.Maintenance_Req."9" := FALSE;   // AC1.Sign.Maintenance_Req.9 > Maintenance 9 request
   Sign.Maintenance_Req."10" := FALSE;   // AC1.Sign.Maintenance_Req.10
   Sign.Maintenance_Req."11" := FALSE;   // AC1.Sign.Maintenance_Req.11
   Sign.Maintenance_Req."12" := FALSE;   // AC1.Sign.Maintenance_Req.12
   Sign.Maintenance_Req."13" := FALSE;   // AC1.Sign.Maintenance_Req.13
   Sign.Maintenance_Req."14" := FALSE;   // AC1.Sign.Maintenance_Req.14
   Sign.Maintenance_Req."15" := FALSE;   // AC1.Sign.Maintenance_Req.15
   Sign.Maintenance_Req."16" := FALSE;   // AC1.Sign.Maintenance_Req.16
   Sign.Maintenance_Req."17" := FALSE;   // AC1.Sign.Maintenance_Req.17
   Sign.Maintenance_Req."18" := FALSE;   // AC1.Sign.Maintenance_Req.18
   Sign.Maintenance_Req."19" := FALSE;   // AC1.Sign.Maintenance_Req.19
   Sign.Maintenance_Req."20" := FALSE;   // AC1.Sign.Maintenance_Req.20
   Sign.Maintenance_Req."21" := FALSE;   // AC1.Sign.Maintenance_Req.21
   Sign.Maintenance_Req."22" := FALSE;   // AC1.Sign.Maintenance_Req.22
   Sign.Maintenance_Req."23" := FALSE;   // AC1.Sign.Maintenance_Req.23
   Sign.Maintenance_Req."24" := FALSE;   // AC1.Sign.Maintenance_Req.24
   Sign.Maintenance_Req."25" := FALSE;   // AC1.Sign.Maintenance_Req.25
   Sign.Maintenance_Req."26" := FALSE;   // AC1.Sign.Maintenance_Req.26
   Sign.Maintenance_Req."27" := FALSE;   // AC1.Sign.Maintenance_Req.27
   Sign.Maintenance_Req."28" := FALSE;   // AC1.Sign.Maintenance_Req.28
   Sign.Maintenance_Req."29" := FALSE;   // AC1.Sign.Maintenance_Req.29
   Sign.Maintenance_Req."30" := FALSE;   // AC1.Sign.Maintenance_Req.30
   Sign.Maintenance_Req."31" := FALSE;   // AC1.Sign.Maintenance_Req.31
   Sign.Maintenance_Activated."0" := FALSE;   // AC1.Sign.Maintenance_Activated.0 > Maintenance 0 activated
   Sign.Maintenance_Activated."1" := FALSE;   // AC1.Sign.Maintenance_Activated.1 > Maintenance 1 activated
   Sign.Maintenance_Activated."2" := FALSE;   // AC1.Sign.Maintenance_Activated.2 > Maintenance 2 activated
   Sign.Maintenance_Activated."3" := FALSE;   // AC1.Sign.Maintenance_Activated.3 > Maintenance 3 activated
   Sign.Maintenance_Activated."4" := FALSE;   // AC1.Sign.Maintenance_Activated.4 > Maintenance 4 activated
   Sign.Maintenance_Activated."5" := FALSE;   // AC1.Sign.Maintenance_Activated.5 > Maintenance 5 activated
   Sign.Maintenance_Activated."6" := FALSE;   // AC1.Sign.Maintenance_Activated.6 > Maintenance 6 activated
   Sign.Maintenance_Activated."7" := FALSE;   // AC1.Sign.Maintenance_Activated.7 > Maintenance 7 activated
   Sign.Maintenance_Activated."8" := FALSE;   // AC1.Sign.Maintenance_Activated.8 > Maintenance 8 activated
   Sign.Maintenance_Activated."9" := FALSE;   // AC1.Sign.Maintenance_Activated.9 > Maintenance 9 activated
   Sign.Maintenance_Activated."10" := FALSE;   // AC1.Sign.Maintenance_Activated.10
   Sign.Maintenance_Activated."11" := FALSE;   // AC1.Sign.Maintenance_Activated.11
   Sign.Maintenance_Activated."12" := FALSE;   // AC1.Sign.Maintenance_Activated.12
   Sign.Maintenance_Activated."13" := FALSE;   // AC1.Sign.Maintenance_Activated.13
   Sign.Maintenance_Activated."14" := FALSE;   // AC1.Sign.Maintenance_Activated.14
   Sign.Maintenance_Activated."15" := FALSE;   // AC1.Sign.Maintenance_Activated.15
   Sign.Maintenance_Activated."16" := FALSE;   // AC1.Sign.Maintenance_Activated.16
   Sign.Maintenance_Activated."17" := FALSE;   // AC1.Sign.Maintenance_Activated.17
   Sign.Maintenance_Activated."18" := FALSE;   // AC1.Sign.Maintenance_Activated.18
   Sign.Maintenance_Activated."19" := FALSE;   // AC1.Sign.Maintenance_Activated.19
   Sign.Maintenance_Activated."20" := FALSE;   // AC1.Sign.Maintenance_Activated.20
   Sign.Maintenance_Activated."21" := FALSE;   // AC1.Sign.Maintenance_Activated.21
   Sign.Maintenance_Activated."22" := FALSE;   // AC1.Sign.Maintenance_Activated.22
   Sign.Maintenance_Activated."23" := FALSE;   // AC1.Sign.Maintenance_Activated.23
   Sign.Maintenance_Activated."24" := FALSE;   // AC1.Sign.Maintenance_Activated.24
   Sign.Maintenance_Activated."25" := FALSE;   // AC1.Sign.Maintenance_Activated.25
   Sign.Maintenance_Activated."26" := FALSE;   // AC1.Sign.Maintenance_Activated.26
   Sign.Maintenance_Activated."27" := FALSE;   // AC1.Sign.Maintenance_Activated.27
   Sign.Maintenance_Activated."28" := FALSE;   // AC1.Sign.Maintenance_Activated.28
   Sign.Maintenance_Activated."29" := FALSE;   // AC1.Sign.Maintenance_Activated.29
   Sign.Maintenance_Activated."30" := FALSE;   // AC1.Sign.Maintenance_Activated.30
   Sign.Maintenance_Activated."31" := FALSE;   // AC1.Sign.Maintenance_Activated.31
   Input.MouPreBtwAscDesc := FALSE;
   Input.InfMouOnLug_OpeSid := TRUE;
   Input.InfMouOnLug_NotOpeSid := FALSE;
   Input.OufMouOnLug_OpeSid := TRUE;
   Input.OufMouOnLug_NotOpeSid := FALSE;
   Input.MouOveTra := FALSE;
   Input.Jog_Rst := FALSE;
   Input.Jog_Cnn := FALSE;
   Input.Jog_Req := FALSE;
   Input.BrkPwrSrvVlv := TRUE;
   Input.BrkPwrFanPmp := TRUE;
   Input.StaPbt := FALSE;
   Input.StoPbt := FALSE;
   Input.RstPbt := FALSE;
   Input.EnaPbt := FALSE;
   Input.Jog_Bit := 0;
   Input.Safety.SafeZone1Ok := TRUE;
   Input.Safety.SafeZone2Ok := FALSE;
   Input.Safety.EmgJog1 := FALSE;
   Input.Safety.DeadMan1 := FALSE;
   Input.Safety.EmgJog2 := FALSE;
   Input.Safety.DeadMan2 := FALSE;
   Input.Safety.DeadMan1Ena := FALSE;
   Input.Safety.DeadMan2Ena := FALSE;
   Input.Safety.SlsAscDesc := FALSE;
   Input.Safety.SlsAsc := FALSE;
   Input.Safety.SlsDesc := FALSE;
   Input.Safety.SlsTra := FALSE;
   Input.Safety.STO_AscDesc := FALSE;
   Input.Safety.STO_Asc := FALSE;
   Input.Safety.STO_Desc := FALSE;
   Input.Safety.STO_Transfer := FALSE;
   Input.Safety.LghCurOpeSid := FALSE;
   Input.Safety.LghCurNotOpeSid := FALSE;
   Input.Safety.Grd_01 := FALSE;
   Input.Safety.Grd_02 := FALSE;
   Input.Safety.Grd_03 := FALSE;
   Input.Safety.Grd_04 := FALSE;
   Input.Safety.Grd_05 := FALSE;
   Input.Safety.Grd_06 := FALSE;
   Input.Safety.Grd_07 := FALSE;
   Input.Safety.Grd_08 := FALSE;
   Input.Safety.Grd_09 := FALSE;
   Input.Safety.Grd_10 := FALSE;
   Input.Safety.SrySen1Trm1InBlk := FALSE;
   Input.Safety.SrySen2Trm1InBlk := FALSE;
   Input.Safety.SrySen1Trm1OutBlk := FALSE;
   Input.Safety.SrySen2Trm1OutBlk := FALSE;
   Input.Safety.QBad_01 := FALSE;
   Input.Safety.QBad_02 := FALSE;
   Input.Safety.QBad_03 := FALSE;
   Input.Safety.QBad_Asc := FALSE;
   Input.Safety.QBad_Desc := FALSE;
   Input.Safety.QBad_AscDesc := FALSE;
   Input.Safety.QBad_Transfer := FALSE;
   Input.Safety.QBad_InvPumpThRgIn1 := FALSE;
   Input.Safety.QBad_InvPumpThRgIn2 := FALSE;
   Input.Safety.QBad_InvPumpThRgOut1 := FALSE;
   Input.Safety.QBad_InvPumpThRgOut2 := FALSE;
   Output.ModLgh := TRUE;
   Ons.TimeWork := TRUE;
   Ons.ShiftAscDesc := FALSE;
   Ons.ShiftTransfer := FALSE;
   Ons.PosOkAscDesc := TRUE;
   Ons.InputSafetyDeadMan := FALSE;
   Ons.ShiftAsc := TRUE;
   Ons.ShiftDesc := TRUE;
   Ons._7 := FALSE;
   Ons._8 := FALSE;
   Ons._9 := FALSE;
   Ons._10 := FALSE;
   Ons._11 := FALSE;
   Ons._12 := FALSE;
   Ons._13 := FALSE;
   Ons._14 := FALSE;
   Ons._15 := FALSE;
   "Step"._00_CycleActivate_StartAscDesc := FALSE;
   "Step"._10_VirtualMasterInMotion := FALSE;
   "Step"._20_AscDescInMotion := FALSE;
   "Step"._30_AscDescDone := FALSE;
   "Step"._40_CycleFinish := FALSE;
   "Step".ScSeqOk := FALSE;
   CamCalc.CalcReq := FALSE;
   CamCalc.OnsCalcReq := FALSE;
   CamCalc.Asc_LenghtUsed := 8;
   CamCalc.Desc_LenghtUsed := 5;
   CamCalc.Transfer_LenghtUsed := 10;
   CamCalc.Asc_Cam[0].leadingValueStart := 0.0;
   CamCalc.Asc_Cam[1].leadingValueStart := 50.0;
   CamCalc.Asc_Cam[2].leadingValueStart := 50.01;
   CamCalc.Asc_Cam[3].leadingValueStart := 100.0;
   CamCalc.Asc_Cam[4].leadingValueStart := 360.0;
   CamCalc.Asc_Cam[5].leadingValueStart := 410.0;
   CamCalc.Asc_Cam[6].leadingValueStart := 410.01;
   CamCalc.Asc_Cam[7].leadingValueStart := 460.0;
   CamCalc.Asc_Cam[8..39].leadingValueStart := 0.0;
   CamCalc.Asc_Cam[0].leadingValueEnd := 50.0;
   CamCalc.Asc_Cam[1].leadingValueEnd := 50.01;
   CamCalc.Asc_Cam[2].leadingValueEnd := 100.0;
   CamCalc.Asc_Cam[3].leadingValueEnd := 360.0;
   CamCalc.Asc_Cam[4].leadingValueEnd := 410.0;
   CamCalc.Asc_Cam[5].leadingValueEnd := 410.01;
   CamCalc.Asc_Cam[6].leadingValueEnd := 460.0;
   CamCalc.Asc_Cam[7].leadingValueEnd := 720.0;
   CamCalc.Asc_Cam[8..39].leadingValueEnd := 0.0;
   CamCalc.Asc_Cam[0].followingValueStart := 0.0;
   CamCalc.Asc_Cam[1].followingValueStart := 28.5750007629395;
   CamCalc.Asc_Cam[2].followingValueStart := 28.5864307632446;
   CamCalc.Asc_Cam[3..4].followingValueStart := 57.1500015258789;
   CamCalc.Asc_Cam[5].followingValueStart := 85.7250022888184;
   CamCalc.Asc_Cam[6].followingValueStart := 85.7364322891235;
   CamCalc.Asc_Cam[7].followingValueStart := 114.300003051758;
   CamCalc.Asc_Cam[8..39].followingValueStart := 0.0;
   CamCalc.Asc_Cam[0].followingValueEnd := 28.5750007629395;
   CamCalc.Asc_Cam[1].followingValueEnd := 28.5864307632446;
   CamCalc.Asc_Cam[2..3].followingValueEnd := 57.1500015258789;
   CamCalc.Asc_Cam[4].followingValueEnd := 85.7250022888184;
   CamCalc.Asc_Cam[5].followingValueEnd := 85.7364322891235;
   CamCalc.Asc_Cam[6..7].followingValueEnd := 114.300003051758;
   CamCalc.Asc_Cam[8..39].followingValueEnd := 0.0;
   CamCalc.Asc_Cam[0].geoVeloStart := 0.0;
   CamCalc.Asc_Cam[1..2].geoVeloStart := 1.14300003051758;
   CamCalc.Asc_Cam[3..4].geoVeloStart := 0.0;
   CamCalc.Asc_Cam[5..6].geoVeloStart := 1.14300003051758;
   CamCalc.Asc_Cam[7..39].geoVeloStart := 0.0;
   CamCalc.Asc_Cam[0..1].geoVeloEnd := 1.14300003051758;
   CamCalc.Asc_Cam[2..3].geoVeloEnd := 0.0;
   CamCalc.Asc_Cam[4..5].geoVeloEnd := 1.14300003051758;
   CamCalc.Asc_Cam[6..39].geoVeloEnd := 0.0;
   CamCalc.Asc_Cam[0..39].geoAccelStart := 0.0;
   CamCalc.Asc_Cam[0..39].geoAccelEnd := 0.0;
   CamCalc.Asc_Cam[0..39].geoJerkStart := 0.0;
   CamCalc.Asc_Cam[0..39].geoJerkEnd := 0.0;
   CamCalc.Asc_Cam[0..39].inflectionPointParameter := 0.5;
   CamCalc.Asc_Cam[0..39].modVeloTrapezoidParameter := 1.0;
   CamCalc.Asc_Cam[0..39].modSineMaxAccelCaStar := 0.0;
   CamCalc.Asc_Cam[0].camProfileType := 4;
   CamCalc.Asc_Cam[1].camProfileType := 3;
   CamCalc.Asc_Cam[2].camProfileType := 4;
   CamCalc.Asc_Cam[3].camProfileType := 2;
   CamCalc.Asc_Cam[4].camProfileType := 4;
   CamCalc.Asc_Cam[5].camProfileType := 3;
   CamCalc.Asc_Cam[6].camProfileType := 4;
   CamCalc.Asc_Cam[7].camProfileType := 2;
   CamCalc.Asc_Cam[8..39].camProfileType := 0;
   CamCalc.Desc_Cam[0].leadingValueStart := 0.0;
   CamCalc.Desc_Cam[1].leadingValueStart := 360.0;
   CamCalc.Desc_Cam[2].leadingValueStart := 410.0;
   CamCalc.Desc_Cam[3].leadingValueStart := 410.01;
   CamCalc.Desc_Cam[4].leadingValueStart := 460.0;
   CamCalc.Desc_Cam[5..39].leadingValueStart := 0.0;
   CamCalc.Desc_Cam[0].leadingValueEnd := 360.0;
   CamCalc.Desc_Cam[1].leadingValueEnd := 410.0;
   CamCalc.Desc_Cam[2].leadingValueEnd := 410.01;
   CamCalc.Desc_Cam[3].leadingValueEnd := 460.0;
   CamCalc.Desc_Cam[4].leadingValueEnd := 720.0;
   CamCalc.Desc_Cam[5..39].leadingValueEnd := 0.0;
   CamCalc.Desc_Cam[0..1].followingValueStart := 0.0;
   CamCalc.Desc_Cam[2].followingValueStart := 28.5750007629395;
   CamCalc.Desc_Cam[3].followingValueStart := 28.5864307632446;
   CamCalc.Desc_Cam[4].followingValueStart := 57.1500015258789;
   CamCalc.Desc_Cam[5..39].followingValueStart := 0.0;
   CamCalc.Desc_Cam[0].followingValueEnd := 0.0;
   CamCalc.Desc_Cam[1].followingValueEnd := 28.5750007629395;
   CamCalc.Desc_Cam[2].followingValueEnd := 28.5864307632446;
   CamCalc.Desc_Cam[3..4].followingValueEnd := 57.1500015258789;
   CamCalc.Desc_Cam[5..39].followingValueEnd := 0.0;
   CamCalc.Desc_Cam[0..1].geoVeloStart := 0.0;
   CamCalc.Desc_Cam[2..3].geoVeloStart := 1.14300003051758;
   CamCalc.Desc_Cam[4..39].geoVeloStart := 0.0;
   CamCalc.Desc_Cam[0].geoVeloEnd := 0.0;
   CamCalc.Desc_Cam[1..2].geoVeloEnd := 1.14300003051758;
   CamCalc.Desc_Cam[3..39].geoVeloEnd := 0.0;
   CamCalc.Desc_Cam[0..39].geoAccelStart := 0.0;
   CamCalc.Desc_Cam[0..39].geoAccelEnd := 0.0;
   CamCalc.Desc_Cam[0..39].geoJerkStart := 0.0;
   CamCalc.Desc_Cam[0..39].geoJerkEnd := 0.0;
   CamCalc.Desc_Cam[0..39].inflectionPointParameter := 0.5;
   CamCalc.Desc_Cam[0..39].modVeloTrapezoidParameter := 1.0;
   CamCalc.Desc_Cam[0..39].modSineMaxAccelCaStar := 0.0;
   CamCalc.Desc_Cam[0].camProfileType := 2;
   CamCalc.Desc_Cam[1].camProfileType := 4;
   CamCalc.Desc_Cam[2].camProfileType := 3;
   CamCalc.Desc_Cam[3].camProfileType := 4;
   CamCalc.Desc_Cam[4].camProfileType := 2;
   CamCalc.Desc_Cam[5..39].camProfileType := 0;
   CamCalc.Transfer_Cam[0].leadingValueStart := 0.0;
   CamCalc.Transfer_Cam[1].leadingValueStart := 100.0;
   CamCalc.Transfer_Cam[2].leadingValueStart := 151.25;
   CamCalc.Transfer_Cam[3].leadingValueStart := 253.75;
   CamCalc.Transfer_Cam[4].leadingValueStart := 305.0;
   CamCalc.Transfer_Cam[5].leadingValueStart := 360.0;
   CamCalc.Transfer_Cam[6].leadingValueStart := 460.0;
   CamCalc.Transfer_Cam[7].leadingValueStart := 511.25;
   CamCalc.Transfer_Cam[8].leadingValueStart := 613.75;
   CamCalc.Transfer_Cam[9].leadingValueStart := 665.0;
   CamCalc.Transfer_Cam[10..39].leadingValueStart := 0.0;
   CamCalc.Transfer_Cam[0].leadingValueEnd := 100.0;
   CamCalc.Transfer_Cam[1].leadingValueEnd := 151.25;
   CamCalc.Transfer_Cam[2].leadingValueEnd := 253.75;
   CamCalc.Transfer_Cam[3].leadingValueEnd := 305.0;
   CamCalc.Transfer_Cam[4].leadingValueEnd := 360.0;
   CamCalc.Transfer_Cam[5].leadingValueEnd := 460.0;
   CamCalc.Transfer_Cam[6].leadingValueEnd := 511.25;
   CamCalc.Transfer_Cam[7].leadingValueEnd := 613.75;
   CamCalc.Transfer_Cam[8].leadingValueEnd := 665.0;
   CamCalc.Transfer_Cam[9].leadingValueEnd := 720.0;
   CamCalc.Transfer_Cam[10..39].leadingValueEnd := 0.0;
   CamCalc.Transfer_Cam[0..1].followingValueStart := 0.0;
   CamCalc.Transfer_Cam[2].followingValueStart := 72.7333323160807;
   CamCalc.Transfer_Cam[3].followingValueStart := 363.666661580404;
   CamCalc.Transfer_Cam[4].followingValueStart := 436.399993896484;
   CamCalc.Transfer_Cam[5..6].followingValueStart := 406.399993896484;
   CamCalc.Transfer_Cam[7].followingValueStart := 479.133326212565;
   CamCalc.Transfer_Cam[8].followingValueStart := 770.066655476888;
   CamCalc.Transfer_Cam[9].followingValueStart := 842.799987792969;
   CamCalc.Transfer_Cam[10..39].followingValueStart := 0.0;
   CamCalc.Transfer_Cam[0].followingValueEnd := 0.0;
   CamCalc.Transfer_Cam[1].followingValueEnd := 72.7333323160807;
   CamCalc.Transfer_Cam[2].followingValueEnd := 363.666661580404;
   CamCalc.Transfer_Cam[3].followingValueEnd := 436.399993896484;
   CamCalc.Transfer_Cam[4..5].followingValueEnd := 406.399993896484;
   CamCalc.Transfer_Cam[6].followingValueEnd := 479.133326212565;
   CamCalc.Transfer_Cam[7].followingValueEnd := 770.066655476888;
   CamCalc.Transfer_Cam[8].followingValueEnd := 842.799987792969;
   CamCalc.Transfer_Cam[9].followingValueEnd := 812.799987792969;
   CamCalc.Transfer_Cam[10..39].followingValueEnd := 0.0;
   CamCalc.Transfer_Cam[0..1].geoVeloStart := 0.0;
   CamCalc.Transfer_Cam[2..3].geoVeloStart := 2.83837394404217;
   CamCalc.Transfer_Cam[4..6].geoVeloStart := 0.0;
   CamCalc.Transfer_Cam[7..8].geoVeloStart := 2.83837394404217;
   CamCalc.Transfer_Cam[9..39].geoVeloStart := 0.0;
   CamCalc.Transfer_Cam[0].geoVeloEnd := 0.0;
   CamCalc.Transfer_Cam[1..2].geoVeloEnd := 2.83837394404217;
   CamCalc.Transfer_Cam[3..5].geoVeloEnd := 0.0;
   CamCalc.Transfer_Cam[6..7].geoVeloEnd := 2.83837394404217;
   CamCalc.Transfer_Cam[8..39].geoVeloEnd := 0.0;
   CamCalc.Transfer_Cam[0..39].geoAccelStart := 0.0;
   CamCalc.Transfer_Cam[0..39].geoAccelEnd := 0.0;
   CamCalc.Transfer_Cam[0..39].geoJerkStart := 0.0;
   CamCalc.Transfer_Cam[0..39].geoJerkEnd := 0.0;
   CamCalc.Transfer_Cam[0..39].inflectionPointParameter := 0.5;
   CamCalc.Transfer_Cam[0..39].modVeloTrapezoidParameter := 1.0;
   CamCalc.Transfer_Cam[0..39].modSineMaxAccelCaStar := 0.0;
   CamCalc.Transfer_Cam[0].camProfileType := 2;
   CamCalc.Transfer_Cam[1].camProfileType := 4;
   CamCalc.Transfer_Cam[2].camProfileType := 3;
   CamCalc.Transfer_Cam[3..4].camProfileType := 4;
   CamCalc.Transfer_Cam[5].camProfileType := 2;
   CamCalc.Transfer_Cam[6].camProfileType := 4;
   CamCalc.Transfer_Cam[7].camProfileType := 3;
   CamCalc.Transfer_Cam[8..9].camProfileType := 4;
   CamCalc.Transfer_Cam[10..39].camProfileType := 0;
   ExchangeFromChain.Chain.EnableMove := FALSE;
   ExchangeFromChain.Chain.StrobeWorkReq := FALSE;
   ExchangeFromChain.Chain.StrobeWorkReqMouldBlock := FALSE;
   ExchangeFromChain.Chain.CheckObstruction := TRUE;
   ExchangeFromChain.Chain.MoveInMan := FALSE;
   ExchangeFromChain.Chain.VMasterInPosition := TRUE;
   ExchangeFromChain.Chain.VMasterAtSpeed := TRUE;
   ExchangeFromChain.Chain.Cfg_1Jog_0Move := FALSE;
   ExchangeFromChain.ShiftMoulds_In.PresMould := TRUE;
   ExchangeFromChain.ShiftMoulds_In.WorkedByDP1 := FALSE;
   ExchangeFromChain.ShiftMoulds_In.WorkedByDP2 := FALSE;
   ExchangeFromChain.ShiftMoulds_In.WorkedByDP3 := FALSE;
   ExchangeFromChain.ShiftMoulds_In.WorkedByDP4 := FALSE;
   ExchangeFromChain.ShiftMoulds_In.WorkedByID1 := FALSE;
   ExchangeFromChain.ShiftMoulds_In.WorkedByID2 := FALSE;
   ExchangeFromChain.ShiftMoulds_In.WorkedByID3 := FALSE;
   ExchangeFromChain.ShiftMoulds_In.WorkedByID4 := FALSE;
   ExchangeFromChain.ShiftMoulds_In.WorkedByBF1 := FALSE;
   ExchangeFromChain.ShiftMoulds_In.WorkedByFS1 := FALSE;
   ExchangeFromChain.ShiftMoulds_In.WorkedByCM1 := FALSE;
   ExchangeFromChain.ShiftMoulds_In.WorkedByOM1 := FALSE;
   ExchangeFromChain.ShiftMoulds_In.WorkedByRD1 := FALSE;
   ExchangeFromChain.ShiftMoulds_In.ProductOK := FALSE;
   ExchangeFromChain.ShiftMoulds_In.RejMould := FALSE;
   ExchangeFromChain.ShiftMoulds_In.RejByShellScale := FALSE;
   ExchangeFromChain.ShiftMoulds_In.RejByFillScale := FALSE;
   ExchangeFromChain.ShiftMoulds_In.RejByTotalScale := FALSE;
   ExchangeFromChain.ShiftMoulds_In.RejByChecker := FALSE;
   ExchangeFromChain.ShiftMoulds_In.RejByTimeout := FALSE;
   ExchangeFromChain.ShiftMoulds_In.RejByCycleInterruption := FALSE;
   ExchangeFromChain.ShiftMoulds_In.MarkedByOpe := FALSE;
   ExchangeFromChain.ShiftMoulds_In.OkByPyrometerDP1 := FALSE;
   ExchangeFromChain.ShiftMoulds_In.OkByPyrometerDP2 := FALSE;
   ExchangeFromChain.ShiftMoulds_In.OkByPyrometerDP3 := FALSE;
   ExchangeFromChain.ShiftMoulds_In.OkByPyrometerDP4 := FALSE;
   ExchangeFromChain.ShiftMoulds_In.OkByPyrometerFS1 := FALSE;
   ExchangeFromChain.ShiftMoulds_In.OkByPyrometerCM1 := FALSE;
   ExchangeFromChain.ShiftMoulds_In.BadStarved := FALSE;
   ExchangeFromChain.ShiftMoulds_In.BadBlocked := FALSE;
   ExchangeFromChain.ShiftMoulds_In.DirtyMould := FALSE;
   ExchangeFromChain.ShiftMoulds_In.WeightEmptyMould := 0.0;
   ExchangeFromChain.ShiftMoulds_In.WeightShell := 0.0;
   ExchangeFromChain.ShiftMoulds_In.WeightFill := 0.0;
   ExchangeFromChain.ShiftMoulds_In.WeightEndProduction := 0.0;
   ExchangeFromChain.SetPointSpeed := 10.0;
   ExchangeFromChain.KConv_DegSec := 6.0;
   ExchangeToChain.Work := FALSE;
   ExchangeToChain.OutChainObstruction := TRUE;
   ExchangeToChain.AlmOKImmStopChain := TRUE;
   ExchangeToChain.TimeWork := 1000;
   ExchangeToChain.ShiftMoulds_Out[0..1].PresMould := FALSE;
   ExchangeToChain.ShiftMoulds_Out[0..1].WorkedByDP1 := FALSE;
   ExchangeToChain.ShiftMoulds_Out[0..1].WorkedByDP2 := FALSE;
   ExchangeToChain.ShiftMoulds_Out[0..1].WorkedByDP3 := FALSE;
   ExchangeToChain.ShiftMoulds_Out[0..1].WorkedByDP4 := FALSE;
   ExchangeToChain.ShiftMoulds_Out[0..1].WorkedByID1 := FALSE;
   ExchangeToChain.ShiftMoulds_Out[0..1].WorkedByID2 := FALSE;
   ExchangeToChain.ShiftMoulds_Out[0..1].WorkedByID3 := FALSE;
   ExchangeToChain.ShiftMoulds_Out[0..1].WorkedByID4 := FALSE;
   ExchangeToChain.ShiftMoulds_Out[0..1].WorkedByBF1 := FALSE;
   ExchangeToChain.ShiftMoulds_Out[0..1].WorkedByFS1 := FALSE;
   ExchangeToChain.ShiftMoulds_Out[0..1].WorkedByCM1 := FALSE;
   ExchangeToChain.ShiftMoulds_Out[0..1].WorkedByOM1 := FALSE;
   ExchangeToChain.ShiftMoulds_Out[0..1].WorkedByRD1 := FALSE;
   ExchangeToChain.ShiftMoulds_Out[0..1].ProductOK := FALSE;
   ExchangeToChain.ShiftMoulds_Out[0..1].RejMould := FALSE;
   ExchangeToChain.ShiftMoulds_Out[0..1].RejByShellScale := FALSE;
   ExchangeToChain.ShiftMoulds_Out[0..1].RejByFillScale := FALSE;
   ExchangeToChain.ShiftMoulds_Out[0..1].RejByTotalScale := FALSE;
   ExchangeToChain.ShiftMoulds_Out[0..1].RejByChecker := FALSE;
   ExchangeToChain.ShiftMoulds_Out[0..1].RejByTimeout := FALSE;
   ExchangeToChain.ShiftMoulds_Out[0..1].RejByCycleInterruption := FALSE;
   ExchangeToChain.ShiftMoulds_Out[0..1].MarkedByOpe := FALSE;
   ExchangeToChain.ShiftMoulds_Out[0..1].OkByPyrometerDP1 := FALSE;
   ExchangeToChain.ShiftMoulds_Out[0..1].OkByPyrometerDP2 := FALSE;
   ExchangeToChain.ShiftMoulds_Out[0..1].OkByPyrometerDP3 := FALSE;
   ExchangeToChain.ShiftMoulds_Out[0..1].OkByPyrometerDP4 := FALSE;
   ExchangeToChain.ShiftMoulds_Out[0..1].OkByPyrometerFS1 := FALSE;
   ExchangeToChain.ShiftMoulds_Out[0..1].OkByPyrometerCM1 := FALSE;
   ExchangeToChain.ShiftMoulds_Out[0..1].BadStarved := FALSE;
   ExchangeToChain.ShiftMoulds_Out[0..1].BadBlocked := FALSE;
   ExchangeToChain.ShiftMoulds_Out[0..1].DirtyMould := FALSE;
   ExchangeToChain.ShiftMoulds_Out[0..1].WeightEmptyMould := 0.0;
   ExchangeToChain.ShiftMoulds_Out[0..1].WeightShell := 0.0;
   ExchangeToChain.ShiftMoulds_Out[0..1].WeightFill := 0.0;
   ExchangeToChain.ShiftMoulds_Out[0..1].WeightEndProduction := 0.0;
   Asc.PosOK := TRUE;
   Asc.PosOKHalf := FALSE;
   Asc.EnMove := FALSE;
   Asc.OkToStop := TRUE;
   Asc.Strobe := FALSE;
   Asc.StrobeShift := FALSE;
   Asc.HalfUnwind := 57.15;
   Asc.TON_DelaySls.PT := T#1S;
   Asc.TON_DelaySls.IN := FALSE;
   Asc.Man.EnaPbt := FALSE;
   Asc.Man.RstCmd := TRUE;
   Asc.Man.ScreenNumber := 304_010_301;
   Asc.Man.WithinScreenRange := 0;
   Asc.Drive.AlmOk := TRUE;
   Asc.Drive.AlmEmerg := FALSE;
   Asc.Drive.AlmNode := FALSE;
   Asc.Drive.InitPosDrive := FALSE;
   Asc.Drive.InitPosDrivePLS := FALSE;
   Asc.Drive.GearingON := FALSE;
   Asc.Drive.CamHook := FALSE;
   Asc.Drive.CamStoppingPhase := FALSE;
   Asc.Drive.RepositioningRequest := FALSE;
   Asc.Drive.CamRequestResult := FALSE;
   Asc.Drive.CamRequestError := FALSE;
   Asc.Drive.CamRequestOk := TRUE;
   Asc.Drive.CalibDisAxisReq := FALSE;
   Asc.Drive.CalibReq := FALSE;
   Asc.Drive.CalibProcess := FALSE;
   Asc.Drive.HwOvertravelDisReq := FALSE;
   Asc.Drive.HwOvertravelEnReq := FALSE;
   Asc.Drive.AuxCamRequest := FALSE;
   Asc.Drive.TorquePeakEna := TRUE;
   Asc.Drive.Cmd_Repos := FALSE;
   Asc.Drive.Ons_CamRequest := FALSE;
   Asc.Drive.AuxCmdPosition := 0;
   Asc.Drive.Unwind := 114.3;
   Asc.Drive.MaxDev := 15.0;
   Asc.Drive.ReposSpeed := 10.0;
   Asc.Drive.CalcSlaveDifferenceABS := 114.299;
   Asc.Drive.CalcModPosition := 0.0;
   Asc.Drive.CalcSlaveDifference := -114.299;
   Asc.Drive.CalcMinDeltaPos := 99.3;
   Asc.Drive.CalcMaxDeltaPos := 15.0;
   Asc.Drive.CalcHalfPosUnwind := 57.15;
   Asc.Drive.Man.Cmd_PosJog := FALSE;
   Asc.Drive.Man.Cmd_NegJog := FALSE;
   Asc.Drive.Man.Cmd_Step := FALSE;
   Asc.Drive.Man.Cmd_Forward := FALSE;
   Asc.Drive.Man.Cmd_Backward := FALSE;
   Asc.Drive.Man.Cmd_Up := FALSE;
   Asc.Drive.Man.Cmd_Down := FALSE;
   Asc.Drive.Man.Cmd_Intermediate := FALSE;
   Asc.Drive.Man.Cmd_Open := FALSE;
   Asc.Drive.Man.Cmd_Close := FALSE;
   Asc.Drive.Man.Cmd_PreOpen := FALSE;
   Asc.Drive.Man.Cmd_Maintenance := FALSE;
   Asc.Drive.Man.Cmd_OperatorSide := FALSE;
   Asc.Drive.Man.Cmd_NotOperatorSide := FALSE;
   Asc.Drive.Man.Cmd_OnMould := FALSE;
   Asc.Drive.Man.Cmd_OffMould := FALSE;
   Asc.Drive.Man.Cmd_Pos0 := FALSE;
   Asc.Drive.Man.Cmd_Pos1 := FALSE;
   Asc.Drive.Man.Cmd_Pos2 := FALSE;
   Asc.Drive.Man.Cmd_Pos3 := FALSE;
   Asc.Drive.Man.Cmd_Pos4 := FALSE;
   Asc.Drive.Man.Cmd_Pos5 := FALSE;
   Asc.Drive.Man.Ons_Step := FALSE;
   Asc.Drive.Man.PhaseJogCmd := TRUE;
   Asc.Drive.Man.CmdStartStep := FALSE;
   Asc.Drive.Man.CmdEndStep := FALSE;
   Asc.Drive.Man.StepCond := FALSE;
   Asc.Drive.Man.TON_DelayHomeCmd.PT := T#3S;
   Asc.Drive.Man.TON_DelayHomeCmd.IN := FALSE;
   Asc.Drive.Auto.Cmd_Step := FALSE;
   Asc.Drive.Auto.Cmd_StartStep := FALSE;
   Asc.Drive.Auto.Cmd_EndStep := FALSE;
   Asc.Drive.Auto.Cmd_Forward := FALSE;
   Asc.Drive.Auto.Cmd_Backward := FALSE;
   Asc.Drive.Auto.Cmd_Up := FALSE;
   Asc.Drive.Auto.Cmd_Down := FALSE;
   Asc.Drive.Auto.Cmd_Intermediate := FALSE;
   Asc.Drive.Auto.Cmd_Open := FALSE;
   Asc.Drive.Auto.Cmd_Close := FALSE;
   Asc.Drive.Auto.Cmd_PreOpen := FALSE;
   Asc.Drive.Auto.Cmd_Maintenance := FALSE;
   Asc.Drive.Auto.Cmd_OperatorSide := FALSE;
   Asc.Drive.Auto.Cmd_NotOperatorSide := FALSE;
   Asc.Drive.Auto.Cmd_OnMould := FALSE;
   Asc.Drive.Auto.Cmd_OffMould := FALSE;
   Asc.Drive.Auto.Cmd_Pos0 := FALSE;
   Asc.Drive.Auto.Cmd_Pos1 := FALSE;
   Asc.Drive.Auto.Cmd_Pos2 := FALSE;
   Asc.Drive.Auto.Cmd_Pos3 := FALSE;
   Asc.Drive.Auto.Cmd_Pos4 := FALSE;
   Asc.Drive.Auto.Cmd_Pos5 := FALSE;
   Asc.Drive.Auto.Cmd_Gear := FALSE;
   Asc.Drive.ACT.CMD.Enable := FALSE;
   Asc.Drive.ACT.CMD.Pos_Mode := FALSE;
   Asc.Drive.ACT.CMD.MergeDisabled := FALSE;
   Asc.Drive.ACT.CMD.SCurve := FALSE;
   Asc.Drive.ACT.CMD.Cam_Mode := TRUE;
   Asc.Drive.ACT.CMD.Cam_Request := FALSE;
   Asc.Drive.ACT.CMD.Cam_PhaseStop := FALSE;
   Asc.Drive.ACT.CMD.Gear_Mode := FALSE;
   Asc.Drive.ACT.CMD.Repos_Req := FALSE;
   Asc.Drive.ACT.CMD.Jog_Pos := FALSE;
   Asc.Drive.ACT.CMD.Jog_Neg := FALSE;
   Asc.Drive.ACT.CMD.Stop := FALSE;
   Asc.Drive.ACT.CMD.Calibration_Req := FALSE;
   Asc.Drive.ACT.CMD.Reset := FALSE;
   Asc.Drive.ACT.CMD.RegInput1 := FALSE;
   Asc.Drive.ACT.CMD.Brake_Release := FALSE;
   Asc.Drive.ACT.CMD.HwPosOvertravel_Dis := FALSE;
   Asc.Drive.ACT.CMD.HwNegOvertravel_Dis := FALSE;
   Asc.Drive.ACT.CMD.HwOvertravel_MSG_En := FALSE;
   Asc.Drive.ACT.CMD.OneShootMove := FALSE;
   Asc.Drive.ACT.CMD.Move_Type := 3;
   Asc.Drive.ACT.CMD.Target_Pos := 0.0;
   Asc.Drive.ACT.CMD.Speed := 5.0;
   Asc.Drive.ACT.CMD.Acceleration := 100.0;
   Asc.Drive.ACT.CMD.Deceleration := 100.0;
   Asc.Drive.ACT.CMD.Torque_Limit := 20.0;
   Asc.Drive.ACT.CMD.Gear_Ratio := 0.0;
   Asc.Drive.ACT.CMD.Mccp_Length := 8;
   Asc.Drive.ACT.CMD.Mccp_StartSlope := 0.0;
   Asc.Drive.ACT.CMD.Mccp_EndSlope := 0.0;
   Asc.Drive.ACT.CMD.Mapc_Direction := 0;
   Asc.Drive.ACT.CMD.Mapc_SlaveScaling := 1.0;
   Asc.Drive.ACT.CMD.Mapc_MasterScaling := 1.0;
   Asc.Drive.ACT.CMD.Mapc_MasterLockPosition := 0.0;
   Asc.Drive.ACT.CMD.Mapc_CamLockPosition := 0.0;
   Asc.Drive.ACT.CMD.Cam[0].leadingValueStart := 0.0;
   Asc.Drive.ACT.CMD.Cam[1].leadingValueStart := 50.0;
   Asc.Drive.ACT.CMD.Cam[2].leadingValueStart := 50.01;
   Asc.Drive.ACT.CMD.Cam[3].leadingValueStart := 100.0;
   Asc.Drive.ACT.CMD.Cam[4].leadingValueStart := 360.0;
   Asc.Drive.ACT.CMD.Cam[5].leadingValueStart := 410.0;
   Asc.Drive.ACT.CMD.Cam[6].leadingValueStart := 410.01;
   Asc.Drive.ACT.CMD.Cam[7].leadingValueStart := 460.0;
   Asc.Drive.ACT.CMD.Cam[8..39].leadingValueStart := 0.0;
   Asc.Drive.ACT.CMD.Cam[0].leadingValueEnd := 50.0;
   Asc.Drive.ACT.CMD.Cam[1].leadingValueEnd := 50.01;
   Asc.Drive.ACT.CMD.Cam[2].leadingValueEnd := 100.0;
   Asc.Drive.ACT.CMD.Cam[3].leadingValueEnd := 360.0;
   Asc.Drive.ACT.CMD.Cam[4].leadingValueEnd := 410.0;
   Asc.Drive.ACT.CMD.Cam[5].leadingValueEnd := 410.01;
   Asc.Drive.ACT.CMD.Cam[6].leadingValueEnd := 460.0;
   Asc.Drive.ACT.CMD.Cam[7].leadingValueEnd := 720.0;
   Asc.Drive.ACT.CMD.Cam[8..39].leadingValueEnd := 0.0;
   Asc.Drive.ACT.CMD.Cam[0].followingValueStart := 0.0;
   Asc.Drive.ACT.CMD.Cam[1].followingValueStart := 28.5750007629395;
   Asc.Drive.ACT.CMD.Cam[2].followingValueStart := 28.5864307632446;
   Asc.Drive.ACT.CMD.Cam[3..4].followingValueStart := 57.1500015258789;
   Asc.Drive.ACT.CMD.Cam[5].followingValueStart := 85.7250022888184;
   Asc.Drive.ACT.CMD.Cam[6].followingValueStart := 85.7364322891235;
   Asc.Drive.ACT.CMD.Cam[7].followingValueStart := 114.300003051758;
   Asc.Drive.ACT.CMD.Cam[8..39].followingValueStart := 0.0;
   Asc.Drive.ACT.CMD.Cam[0].followingValueEnd := 28.5750007629395;
   Asc.Drive.ACT.CMD.Cam[1].followingValueEnd := 28.5864307632446;
   Asc.Drive.ACT.CMD.Cam[2..3].followingValueEnd := 57.1500015258789;
   Asc.Drive.ACT.CMD.Cam[4].followingValueEnd := 85.7250022888184;
